Yaskawa INFORM job: A_ROOF_UPPER_0614_2_PAINT_44.JBI

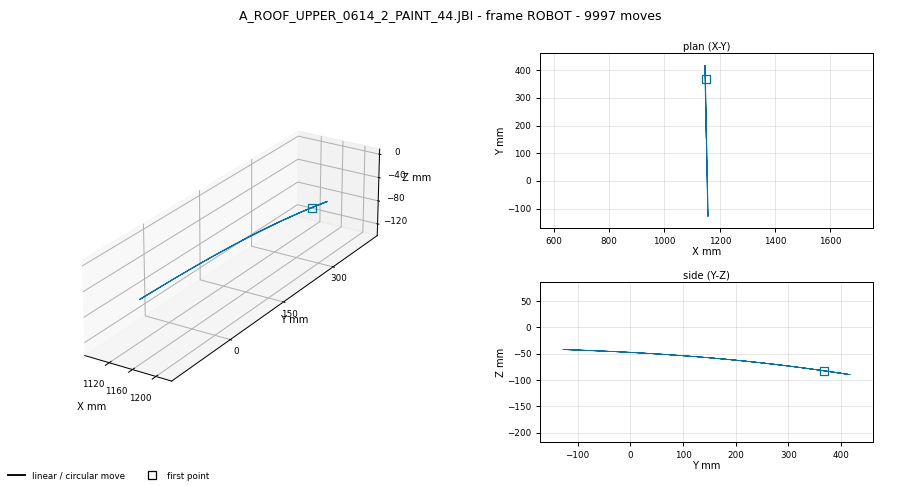
[picture p0: tool path of A_ROOF_UPPER_0614_2_PAINT_44.JBI in frame ROBOT, 9997 of 9997 moves have a stored position in this frame; points joined in program order, loops and branches not executed]
/JOB
//NAME A_ROOF_UPPER_0614_2_PAINT44
//POS
///NPOS 9997,0,0,0,0,0
///TOOL 1
///USER 0
///POSTYPE ROBOT
///RECTAN
///RCONF 1,0,0,0,0,0,0,0,0,0,0,0,0,0,0,0,0,0,0,0,0,0,0,0
C00000=1148.785,367.055,-82.178,-176.274,9.416,148.837
C00001=1148.782,367.302,-82.214,-176.271,9.420,148.837
C00002=1148.778,367.550,-82.249,-176.269,9.424,148.838
C00003=1148.773,367.797,-82.285,-176.266,9.428,148.838
C00004=1148.769,368.045,-82.321,-176.263,9.433,148.839
C00005=1148.766,368.292,-82.356,-176.261,9.436,148.839
C00006=1148.762,368.540,-82.392,-176.258,9.440,148.839
C00007=1148.758,368.787,-82.429,-176.256,9.445,148.840
C00008=1148.754,369.034,-82.464,-176.253,9.449,148.840
C00009=1148.751,369.282,-82.500,-176.250,9.453,148.841
C00010=1148.747,369.529,-82.535,-176.248,9.457,148.841
C00011=1148.742,369.776,-82.571,-176.246,9.461,148.841
C00012=1148.738,370.024,-82.607,-176.243,9.465,148.842
C00013=1148.735,370.271,-82.643,-176.241,9.470,148.842
C00014=1148.731,370.519,-82.679,-176.239,9.473,148.843
C00015=1148.727,370.766,-82.715,-176.236,9.477,148.843
C00016=1148.723,371.014,-82.750,-176.233,9.482,148.843
C00017=1148.719,371.261,-82.787,-176.231,9.486,148.844
C00018=1148.716,371.508,-82.823,-176.228,9.490,148.844
C00019=1148.712,371.756,-82.858,-176.226,9.494,148.845
C00020=1148.708,372.003,-82.895,-176.224,9.498,148.845
C00021=1148.704,372.250,-82.931,-176.221,9.503,148.846
C00022=1148.700,372.498,-82.966,-176.219,9.506,148.846
C00023=1148.696,372.745,-83.003,-176.217,9.510,148.846
C00024=1148.693,372.993,-83.039,-176.214,9.515,148.847
C00025=1148.689,373.240,-83.075,-176.212,9.519,148.847
C00026=1148.684,373.487,-83.111,-176.210,9.523,148.848
C00027=1148.680,373.734,-83.147,-176.208,9.527,148.848
C00028=1148.677,373.981,-83.183,-176.205,9.532,148.849
C00029=1148.673,374.229,-83.219,-176.203,9.535,148.849
C00030=1148.669,374.476,-83.255,-176.201,9.540,148.850
C00031=1148.665,374.724,-83.291,-176.199,9.543,148.850
C00032=1148.661,374.971,-83.328,-176.196,9.548,148.851
C00033=1148.657,375.218,-83.363,-176.194,9.553,148.851
C00034=1148.654,375.466,-83.401,-176.192,9.556,148.852
C00035=1148.651,375.713,-83.437,-176.190,9.561,148.852
C00036=1148.646,375.961,-83.473,-176.188,9.564,148.853
C00037=1148.643,376.208,-83.509,-176.186,9.569,148.853
C00038=1148.638,376.455,-83.545,-176.184,9.573,148.854
C00039=1148.635,376.702,-83.582,-176.182,9.577,148.854
C00040=1148.631,376.950,-83.618,-176.180,9.581,148.855
C00041=1148.627,377.197,-83.655,-176.179,9.585,148.855
C00042=1148.623,377.444,-83.691,-176.177,9.589,148.856
C00043=1148.619,377.692,-83.727,-176.175,9.593,148.856
C00044=1148.615,377.939,-83.763,-176.173,9.597,148.857
C00045=1148.611,378.186,-83.800,-176.171,9.601,148.858
C00046=1148.608,378.434,-83.836,-176.170,9.605,148.858
C00047=1148.604,378.681,-83.873,-176.168,9.609,148.859
C00048=1148.599,378.928,-83.909,-176.166,9.613,148.859
C00049=1148.596,379.175,-83.946,-176.164,9.617,148.860
C00050=1148.592,379.423,-83.982,-176.163,9.621,148.861
C00051=1148.588,379.670,-84.019,-176.161,9.625,148.861
C00052=1148.585,379.917,-84.055,-176.160,9.629,148.862
C00053=1148.581,380.165,-84.092,-176.158,9.633,148.863
C00054=1148.577,380.412,-84.129,-176.157,9.637,148.863
C00055=1148.573,380.659,-84.165,-176.156,9.641,148.864
C00056=1148.569,380.907,-84.201,-176.154,9.645,148.865
C00057=1148.565,381.154,-84.238,-176.153,9.648,148.865
C00058=1148.561,381.401,-84.275,-176.152,9.652,148.866
C00059=1148.557,381.648,-84.311,-176.151,9.656,148.867
C00060=1148.554,381.896,-84.349,-176.149,9.660,148.867
C00061=1148.550,382.143,-84.384,-176.149,9.663,148.868
C00062=1148.546,382.390,-84.421,-176.147,9.667,148.869
C00063=1148.542,382.638,-84.458,-176.147,9.671,148.869
C00064=1148.539,382.884,-84.494,-176.145,9.675,148.870
C00065=1148.535,383.132,-84.531,-176.145,9.678,148.871
C00066=1148.531,383.379,-84.568,-176.144,9.682,148.871
C00067=1148.527,383.627,-84.605,-176.143,9.685,148.872
C00068=1148.524,383.874,-84.641,-176.142,9.689,148.873
C00069=1148.520,384.121,-84.678,-176.142,9.692,148.874
C00070=1148.515,384.368,-84.715,-176.141,9.696,148.874
C00071=1148.511,384.615,-84.752,-176.140,9.700,148.875
C00072=1148.508,384.862,-84.788,-176.140,9.703,148.876
C00073=1148.505,385.110,-84.825,-176.139,9.706,148.877
C00074=1148.500,385.357,-84.862,-176.140,9.709,148.877
C00075=1148.496,385.604,-84.899,-176.139,9.712,148.878
C00076=1148.493,385.851,-84.935,-176.139,9.716,148.879
C00077=1148.489,386.098,-84.972,-176.138,9.719,148.880
C00078=1148.485,386.346,-85.009,-176.139,9.722,148.881
C00079=1148.481,386.593,-85.046,-176.138,9.725,148.881
C00080=1148.477,386.841,-85.083,-176.139,9.728,148.882
C00081=1148.474,387.088,-85.119,-176.138,9.732,148.883
C00082=1148.470,387.335,-85.156,-176.138,9.734,148.884
C00083=1148.466,387.583,-85.194,-176.138,9.738,148.885
C00084=1148.462,387.830,-85.230,-176.138,9.740,148.885
C00085=1148.458,388.077,-85.267,-176.139,9.743,148.886
C00086=1148.455,388.324,-85.304,-176.139,9.746,148.887
C00087=1148.451,388.571,-85.340,-176.139,9.749,148.888
C00088=1148.447,388.819,-85.378,-176.139,9.752,148.889
C00089=1148.443,389.066,-85.414,-176.140,9.755,148.889
C00090=1148.439,389.313,-85.451,-176.140,9.758,148.890
C00091=1148.436,389.560,-85.488,-176.141,9.761,148.891
C00092=1148.431,389.807,-85.524,-176.141,9.763,148.892
C00093=1148.428,390.055,-85.562,-176.141,9.766,148.893
C00094=1148.424,390.302,-85.599,-176.142,9.769,148.894
C00095=1148.420,390.549,-85.636,-176.143,9.771,148.895
C00096=1148.416,390.836,-85.678,-176.143,9.774,148.895
C00097=1148.411,391.123,-85.721,-176.144,9.777,148.896
C00098=1148.407,391.409,-85.764,-176.145,9.780,148.897
C00099=1148.402,391.696,-85.807,-176.145,9.783,148.898
C00100=1148.399,391.943,-85.843,-176.146,9.786,148.899
C00101=1148.395,392.190,-85.881,-176.146,9.789,148.900
C00102=1148.391,392.437,-85.918,-176.148,9.791,148.901
C00103=1148.387,392.684,-85.955,-176.148,9.793,148.902
C00104=1148.384,392.932,-85.992,-176.149,9.795,148.902
C00105=1148.380,393.179,-86.029,-176.149,9.798,148.903
C00106=1148.376,393.426,-86.065,-176.150,9.800,148.904
C00107=1148.372,393.674,-86.102,-176.151,9.802,148.905
C00108=1148.368,393.921,-86.139,-176.152,9.805,148.906
C00109=1148.365,394.168,-86.177,-176.153,9.807,148.907
C00110=1148.361,394.415,-86.214,-176.154,9.809,148.908
C00111=1148.357,394.662,-86.250,-176.155,9.812,148.909
C00112=1148.353,394.910,-86.287,-176.156,9.814,148.909
C00113=1148.350,395.157,-86.324,-176.157,9.816,148.910
C00114=1148.346,395.404,-86.361,-176.158,9.818,148.911
C00115=1148.342,395.652,-86.398,-176.159,9.821,148.912
C00116=1148.338,395.899,-86.435,-176.160,9.823,148.913
C00117=1148.334,396.146,-86.472,-176.160,9.825,148.913
C00118=1148.330,396.393,-86.509,-176.161,9.827,148.914
C00119=1148.326,396.640,-86.546,-176.163,9.829,148.915
C00120=1148.322,396.888,-86.583,-176.164,9.831,148.916
C00121=1148.319,397.134,-86.619,-176.165,9.833,148.917
C00122=1148.315,397.382,-86.657,-176.165,9.836,148.918
C00123=1148.311,397.630,-86.693,-176.166,9.838,148.918
C00124=1148.307,397.876,-86.731,-176.167,9.840,148.919
C00125=1148.303,398.123,-86.768,-176.169,9.842,148.920
C00126=1148.300,398.371,-86.805,-176.170,9.844,148.921
C00127=1148.296,398.618,-86.842,-176.171,9.846,148.922
C00128=1148.292,398.865,-86.878,-176.172,9.848,148.923
C00129=1148.288,399.112,-86.915,-176.173,9.851,148.924
C00130=1148.284,399.360,-86.952,-176.174,9.852,148.924
C00131=1148.281,399.607,-86.990,-176.175,9.854,148.925
C00132=1148.277,399.854,-87.027,-176.176,9.856,148.926
C00133=1148.273,400.101,-87.064,-176.177,9.858,148.927
C00134=1148.269,400.348,-87.100,-176.179,9.860,148.927
C00135=1148.265,400.596,-87.138,-176.180,9.862,148.928
C00136=1148.262,400.843,-87.174,-176.181,9.864,148.929
C00137=1148.258,401.090,-87.211,-176.182,9.866,148.930
C00138=1148.254,401.337,-87.248,-176.183,9.868,148.931
C00139=1148.251,401.585,-87.286,-176.184,9.870,148.931
C00140=1148.246,401.832,-87.322,-176.185,9.872,148.932
C00141=1148.242,402.079,-87.359,-176.186,9.874,148.933
C00142=1148.238,402.326,-87.396,-176.187,9.876,148.934
C00143=1148.234,402.574,-87.433,-176.188,9.878,148.935
C00144=1148.231,402.821,-87.470,-176.189,9.880,148.935
C00145=1148.228,403.068,-87.507,-176.191,9.881,148.936
C00146=1148.224,403.315,-87.544,-176.192,9.883,148.937
C00147=1148.219,403.562,-87.581,-176.192,9.885,148.938
C00148=1148.216,403.810,-87.618,-176.193,9.887,148.939
C00149=1148.212,404.057,-87.655,-176.195,9.889,148.939
C00150=1148.208,404.304,-87.692,-176.195,9.891,148.940
C00151=1148.204,404.551,-87.728,-176.196,9.893,148.941
C00152=1148.201,404.799,-87.766,-176.197,9.895,148.942
C00153=1148.197,405.046,-87.803,-176.198,9.897,148.942
C00154=1148.193,405.293,-87.840,-176.200,9.898,148.943
C00155=1148.189,405.540,-87.877,-176.201,9.900,148.944
C00156=1148.185,405.788,-87.914,-176.202,9.902,148.945
C00157=1148.181,406.035,-87.951,-176.203,9.904,148.945
C00158=1148.177,406.282,-87.988,-176.204,9.906,148.946
C00159=1148.174,406.529,-88.025,-176.204,9.907,148.947
C00160=1148.170,406.776,-88.061,-176.205,9.909,148.948
C00161=1148.167,407.024,-88.099,-176.206,9.911,148.948
C00162=1148.163,407.271,-88.135,-176.207,9.913,148.949
C00163=1148.158,407.518,-88.172,-176.208,9.915,148.950
C00164=1148.154,407.765,-88.209,-176.209,9.917,148.951
C00165=1148.151,408.013,-88.247,-176.210,9.919,148.951
C00166=1148.147,408.260,-88.284,-176.211,9.921,148.952
C00167=1148.144,408.507,-88.320,-176.212,9.922,148.953
C00168=1148.140,408.754,-88.357,-176.213,9.924,148.954
C00169=1148.136,409.002,-88.394,-176.214,9.926,148.954
C00170=1148.132,409.249,-88.431,-176.215,9.928,148.955
C00171=1148.128,409.496,-88.468,-176.216,9.930,148.956
C00172=1148.124,409.743,-88.506,-176.217,9.932,148.956
C00173=1148.121,409.991,-88.543,-176.218,9.934,148.957
C00174=1148.117,410.238,-88.580,-176.218,9.935,148.958
C00175=1148.113,410.485,-88.616,-176.219,9.937,148.959
C00176=1148.109,410.732,-88.653,-176.220,9.939,148.959
C00177=1148.105,410.979,-88.690,-176.221,9.941,148.960
C00178=1148.102,411.226,-88.728,-176.222,9.943,148.961
C00179=1148.098,411.474,-88.764,-176.222,9.946,148.962
C00180=1148.094,411.721,-88.801,-176.223,9.947,148.962
C00181=1148.090,411.968,-88.838,-176.224,9.949,148.963
C00182=1148.086,412.216,-88.875,-176.225,9.951,148.964
C00183=1148.082,412.463,-88.912,-176.225,9.953,148.964
C00184=1148.079,412.709,-88.949,-176.226,9.955,148.965
C00185=1148.075,412.956,-88.986,-176.227,9.957,148.966
C00186=1148.071,413.204,-89.023,-176.228,9.958,148.966
C00187=1148.067,413.452,-89.060,-176.229,9.961,148.967
C00188=1148.063,413.699,-89.097,-176.229,9.962,148.968
C00189=1148.059,413.946,-89.134,-176.229,9.965,148.969
C00190=1148.056,414.193,-89.172,-176.230,9.967,148.969
C00191=1148.052,414.440,-89.209,-176.231,9.969,148.970
C00192=1148.048,414.688,-89.246,-176.232,9.970,148.971
C00193=1148.045,414.935,-89.282,-176.233,9.972,148.971
C00194=1148.042,415.182,-89.320,-176.233,9.974,148.972
C00195=1148.040,415.429,-89.356,-176.234,9.977,148.973
C00196=1148.039,415.660,-89.390,-176.234,9.979,148.974
C00197=1148.039,415.890,-89.424,-176.235,9.980,148.974
C00198=1148.039,416.119,-89.458,-176.235,9.982,148.975
C00199=1148.040,416.350,-89.492,-176.236,9.983,148.975
C00200=1148.042,416.578,-89.526,-176.237,9.985,148.976
C00201=1148.044,416.809,-89.559,-176.237,9.987,148.977
C00202=1148.046,417.039,-89.593,-176.238,9.988,148.977
C00203=1148.050,417.267,-89.627,-176.238,9.990,148.978
C00204=1147.629,417.270,-89.676,-176.241,10.001,148.981
C00205=1147.626,417.038,-89.642,-176.240,9.999,148.980
C00206=1147.623,416.808,-89.609,-176.240,9.998,148.980
C00207=1147.621,416.576,-89.574,-176.239,9.996,148.979
C00208=1147.619,416.345,-89.540,-176.239,9.994,148.979
C00209=1147.619,416.113,-89.506,-176.238,9.992,148.978
C00210=1147.618,415.881,-89.472,-176.237,9.991,148.977
C00211=1147.619,415.649,-89.438,-176.237,9.989,148.977
C00212=1147.620,415.417,-89.403,-176.236,9.987,148.976
C00213=1147.622,415.171,-89.366,-176.235,9.985,148.976
C00214=1147.625,414.923,-89.329,-176.235,9.984,148.975
C00215=1147.627,414.676,-89.293,-176.235,9.981,148.974
C00216=1147.631,414.429,-89.255,-176.233,9.979,148.973
C00217=1147.635,414.182,-89.218,-176.233,9.977,148.973
C00218=1147.639,413.934,-89.181,-176.232,9.976,148.972
C00219=1147.643,413.687,-89.144,-176.231,9.973,148.971
C00220=1147.647,413.440,-89.107,-176.230,9.972,148.971
C00221=1147.651,413.193,-89.070,-176.230,9.969,148.970
C00222=1147.653,412.945,-89.033,-176.230,9.967,148.969
C00223=1147.658,412.698,-88.996,-176.228,9.965,148.968
C00224=1147.662,412.451,-88.960,-176.228,9.964,148.968
C00225=1147.666,412.204,-88.923,-176.227,9.962,148.967
C00226=1147.669,411.956,-88.885,-176.226,9.960,148.966
C00227=1147.673,411.709,-88.848,-176.225,9.958,148.966
C00228=1147.677,411.462,-88.811,-176.224,9.956,148.965
C00229=1147.681,411.215,-88.774,-176.224,9.954,148.964
C00230=1147.685,410.967,-88.737,-176.223,9.952,148.963
C00231=1147.688,410.720,-88.701,-176.222,9.950,148.963
C00232=1147.692,410.473,-88.664,-176.221,9.949,148.962
C00233=1147.696,410.226,-88.626,-176.220,9.947,148.961
C00234=1147.700,409.979,-88.589,-176.219,9.945,148.961
C00235=1147.704,409.731,-88.552,-176.218,9.943,148.960
C00236=1147.708,409.484,-88.515,-176.218,9.941,148.959
C00237=1147.712,409.237,-88.478,-176.217,9.939,148.958
C00238=1147.715,408.990,-88.441,-176.216,9.937,148.958
C00239=1147.719,408.743,-88.404,-176.215,9.935,148.957
C00240=1147.722,408.496,-88.367,-176.214,9.933,148.956
C00241=1147.726,408.248,-88.331,-176.213,9.931,148.955
C00242=1147.731,408.001,-88.294,-176.212,9.930,148.955
C00243=1147.734,407.753,-88.256,-176.211,9.927,148.954
C00244=1147.738,407.507,-88.219,-176.211,9.926,148.953
C00245=1147.742,407.260,-88.182,-176.209,9.924,148.952
C00246=1147.746,407.012,-88.145,-176.208,9.922,148.952
C00247=1147.749,406.765,-88.108,-176.208,9.920,148.951
C00248=1147.753,406.518,-88.072,-176.207,9.918,148.950
C00249=1147.757,406.270,-88.035,-176.206,9.916,148.950
C00250=1147.761,406.024,-87.997,-176.204,9.915,148.949
C00251=1147.764,405.776,-87.960,-176.203,9.913,148.948
C00252=1147.768,405.529,-87.923,-176.202,9.911,148.947
C00253=1147.772,405.282,-87.886,-176.201,9.909,148.946
C00254=1147.777,405.034,-87.849,-176.200,9.907,148.946
C00255=1147.780,404.787,-87.812,-176.200,9.905,148.945
C00256=1147.784,404.539,-87.775,-176.198,9.903,148.944
C00257=1147.787,404.293,-87.738,-176.197,9.901,148.943
C00258=1147.791,404.046,-87.702,-176.196,9.899,148.942
C00259=1147.795,403.799,-87.665,-176.195,9.898,148.942
C00260=1147.799,403.551,-87.627,-176.194,9.896,148.941
C00261=1147.803,403.304,-87.591,-176.193,9.894,148.940
C00262=1147.807,403.056,-87.554,-176.192,9.892,148.939
C00263=1147.811,402.810,-87.516,-176.191,9.890,148.939
C00264=1147.814,402.562,-87.479,-176.190,9.888,148.938
C00265=1147.818,402.315,-87.443,-176.189,9.886,148.937
C00266=1147.822,402.068,-87.406,-176.188,9.884,148.936
C00267=1147.826,401.821,-87.369,-176.187,9.882,148.935
C00268=1147.829,401.573,-87.332,-176.185,9.881,148.935
C00269=1147.833,401.326,-87.294,-176.184,9.879,148.934
C00270=1147.837,401.079,-87.257,-176.183,9.877,148.933
C00271=1147.841,400.832,-87.220,-176.182,9.875,148.932
C00272=1147.845,400.584,-87.183,-176.181,9.873,148.931
C00273=1147.848,400.337,-87.147,-176.180,9.871,148.931
C00274=1147.852,400.090,-87.110,-176.179,9.868,148.930
C00275=1147.856,399.843,-87.072,-176.178,9.867,148.929
C00276=1147.860,399.595,-87.035,-176.177,9.865,148.928
C00277=1147.864,399.348,-86.998,-176.176,9.863,148.927
C00278=1147.868,399.101,-86.962,-176.175,9.861,148.927
C00279=1147.872,398.854,-86.925,-176.174,9.859,148.926
C00280=1147.876,398.607,-86.888,-176.173,9.856,148.925
C00281=1147.879,398.359,-86.851,-176.171,9.854,148.924
C00282=1147.882,398.113,-86.814,-176.170,9.852,148.923
C00283=1147.887,397.865,-86.777,-176.169,9.850,148.922
C00284=1147.891,397.618,-86.740,-176.168,9.848,148.922
C00285=1147.894,397.370,-86.703,-176.167,9.846,148.921
C00286=1147.898,397.123,-86.666,-176.166,9.844,148.920
C00287=1147.902,396.876,-86.629,-176.165,9.842,148.919
C00288=1147.906,396.629,-86.591,-176.164,9.840,148.918
C00289=1147.909,396.382,-86.555,-176.163,9.838,148.918
C00290=1147.913,396.135,-86.518,-176.162,9.836,148.917
C00291=1147.917,395.887,-86.481,-176.161,9.834,148.916
C00292=1147.921,395.640,-86.444,-176.160,9.831,148.915
C00293=1147.925,395.392,-86.407,-176.159,9.829,148.914
C00294=1147.929,395.145,-86.370,-176.158,9.827,148.913
C00295=1147.933,394.899,-86.333,-176.157,9.825,148.913
C00296=1147.937,394.651,-86.296,-176.157,9.822,148.912
C00297=1147.940,394.404,-86.259,-176.155,9.820,148.911
C00298=1147.943,394.157,-86.222,-176.154,9.818,148.910
C00299=1147.948,393.909,-86.185,-176.153,9.816,148.909
C00300=1147.952,393.662,-86.148,-176.153,9.813,148.908
C00301=1147.956,393.415,-86.112,-176.152,9.811,148.907
C00302=1147.959,393.168,-86.074,-176.151,9.808,148.907
C00303=1147.963,392.921,-86.037,-176.150,9.806,148.906
C00304=1147.966,392.674,-86.001,-176.150,9.804,148.905
C00305=1147.970,392.426,-85.964,-176.149,9.801,148.904
C00306=1147.974,392.179,-85.926,-176.148,9.799,148.903
C00307=1147.978,391.931,-85.890,-176.147,9.797,148.902
C00308=1147.982,391.684,-85.853,-176.147,9.794,148.901
C00309=1147.986,391.398,-85.810,-176.146,9.791,148.901
C00310=1147.991,391.111,-85.767,-176.145,9.788,148.900
C00311=1147.996,390.825,-85.724,-176.145,9.785,148.899
C00312=1148.000,390.538,-85.681,-176.144,9.782,148.898
C00313=1148.003,390.290,-85.644,-176.143,9.780,148.897
C00314=1148.007,390.043,-85.608,-176.142,9.777,148.896
C00315=1148.011,389.796,-85.571,-176.142,9.774,148.895
C00316=1148.015,389.549,-85.534,-176.142,9.772,148.894
C00317=1148.018,389.302,-85.496,-176.141,9.769,148.894
C00318=1148.022,389.054,-85.459,-176.141,9.766,148.893
C00319=1148.026,388.807,-85.422,-176.141,9.763,148.892
C00320=1148.030,388.560,-85.386,-176.140,9.760,148.891
C00321=1148.034,388.313,-85.349,-176.140,9.758,148.890
C00322=1148.037,388.065,-85.312,-176.140,9.754,148.889
C00323=1148.041,387.818,-85.275,-176.140,9.752,148.889
C00324=1148.045,387.571,-85.238,-176.139,9.749,148.888
C00325=1148.049,387.324,-85.202,-176.140,9.745,148.887
C00326=1148.053,387.077,-85.165,-176.139,9.742,148.886
C00327=1148.056,386.829,-85.128,-176.139,9.740,148.885
C00328=1148.061,386.582,-85.091,-176.139,9.736,148.884
C00329=1148.065,386.335,-85.054,-176.140,9.733,148.884
C00330=1148.068,386.088,-85.018,-176.140,9.730,148.883
C00331=1148.071,385.840,-84.981,-176.140,9.727,148.882
C00332=1148.076,385.593,-84.944,-176.140,9.723,148.881
C00333=1148.080,385.345,-84.907,-176.140,9.721,148.881
C00334=1148.084,385.098,-84.870,-176.141,9.717,148.880
C00335=1148.087,384.851,-84.834,-176.141,9.714,148.879
C00336=1148.091,384.604,-84.797,-176.142,9.710,148.878
C00337=1148.095,384.356,-84.760,-176.142,9.707,148.878
C00338=1148.099,384.109,-84.723,-176.143,9.704,148.877
C00339=1148.102,383.862,-84.687,-176.144,9.700,148.876
C00340=1148.106,383.615,-84.650,-176.145,9.696,148.875
C00341=1148.110,383.368,-84.613,-176.145,9.693,148.875
C00342=1148.114,383.121,-84.576,-176.146,9.689,148.874
C00343=1148.117,382.873,-84.540,-176.147,9.686,148.873
C00344=1148.121,382.626,-84.503,-176.147,9.682,148.873
C00345=1148.125,382.379,-84.466,-176.149,9.678,148.872
C00346=1148.129,382.131,-84.429,-176.150,9.674,148.871
C00347=1148.133,381.885,-84.393,-176.151,9.671,148.871
C00348=1148.137,381.637,-84.356,-176.152,9.667,148.870
C00349=1148.141,381.389,-84.319,-176.153,9.663,148.869
C00350=1148.144,381.142,-84.283,-176.155,9.659,148.869
C00351=1148.148,380.895,-84.246,-176.155,9.656,148.868
C00352=1148.152,380.648,-84.209,-176.157,9.652,148.867
C00353=1148.156,380.401,-84.173,-176.158,9.648,148.867
C00354=1148.160,380.154,-84.136,-176.160,9.644,148.866
C00355=1148.164,379.906,-84.100,-176.161,9.640,148.865
C00356=1148.167,379.659,-84.064,-176.163,9.636,148.865
C00357=1148.172,379.412,-84.027,-176.164,9.633,148.864
C00358=1148.175,379.164,-83.990,-176.166,9.629,148.863
C00359=1148.178,378.917,-83.954,-176.168,9.624,148.863
C00360=1148.183,378.669,-83.917,-176.169,9.620,148.862
C00361=1148.186,378.422,-83.881,-176.171,9.616,148.862
C00362=1148.190,378.175,-83.844,-176.173,9.613,148.861
C00363=1148.195,377.927,-83.808,-176.175,9.608,148.860
C00364=1148.198,377.680,-83.772,-176.176,9.604,148.860
C00365=1148.202,377.433,-83.735,-176.178,9.600,148.859
C00366=1148.206,377.186,-83.699,-176.180,9.596,148.859
C00367=1148.210,376.938,-83.663,-176.182,9.592,148.858
C00368=1148.214,376.691,-83.626,-176.184,9.588,148.858
C00369=1148.218,376.444,-83.590,-176.186,9.584,148.857
C00370=1148.222,376.197,-83.553,-176.188,9.580,148.857
C00371=1148.225,375.950,-83.517,-176.190,9.576,148.856
C00372=1148.229,375.702,-83.481,-176.192,9.572,148.856
C00373=1148.233,375.455,-83.445,-176.194,9.567,148.855
C00374=1148.237,375.207,-83.409,-176.197,9.563,148.855
C00375=1148.241,374.960,-83.372,-176.199,9.559,148.854
C00376=1148.245,374.712,-83.336,-176.201,9.555,148.854
C00377=1148.248,374.465,-83.299,-176.203,9.551,148.853
C00378=1148.252,374.217,-83.263,-176.205,9.547,148.853
C00379=1148.256,373.970,-83.227,-176.208,9.542,148.852
C00380=1148.260,373.722,-83.191,-176.209,9.539,148.852
C00381=1148.263,373.476,-83.155,-176.212,9.534,148.851
C00382=1148.268,373.229,-83.119,-176.214,9.530,148.851
C00383=1148.272,372.982,-83.083,-176.216,9.526,148.850
C00384=1148.275,372.734,-83.047,-176.219,9.522,148.850
C00385=1148.280,372.486,-83.011,-176.221,9.518,148.849
C00386=1148.283,372.239,-82.975,-176.224,9.513,148.849
C00387=1148.287,371.992,-82.939,-176.226,9.510,148.849
C00388=1148.291,371.745,-82.902,-176.228,9.505,148.848
C00389=1148.294,371.497,-82.867,-176.231,9.501,148.848
C00390=1148.299,371.249,-82.831,-176.233,9.496,148.847
C00391=1148.303,371.002,-82.795,-176.235,9.493,148.847
C00392=1148.306,370.755,-82.759,-176.238,9.489,148.846
C00393=1148.310,370.507,-82.723,-176.240,9.484,148.846
C00394=1148.314,370.260,-82.687,-176.243,9.480,148.845
C00395=1148.317,370.013,-82.651,-176.246,9.476,148.845
C00396=1148.322,369.765,-82.615,-176.248,9.472,148.845
C00397=1148.325,369.517,-82.579,-176.250,9.468,148.844
C00398=1148.330,369.271,-82.544,-176.253,9.464,148.844
C00399=1148.333,369.023,-82.508,-176.256,9.459,148.844
C00400=1148.337,368.776,-82.472,-176.258,9.455,148.843
C00401=1148.341,368.528,-82.436,-176.260,9.452,148.843
C00402=1148.345,368.281,-82.400,-176.263,9.447,148.842
C00403=1148.349,368.033,-82.364,-176.265,9.443,148.842
C00404=1148.353,367.786,-82.329,-176.268,9.439,148.842
C00405=1148.356,367.538,-82.293,-176.271,9.434,148.841
C00406=1148.361,367.291,-82.258,-176.273,9.431,148.841
C00407=1148.364,367.044,-82.222,-176.276,9.427,148.841
C00408=1148.369,366.796,-82.186,-176.279,9.423,148.840
C00409=1148.372,366.549,-82.151,-176.281,9.418,148.840
C00410=1148.376,366.301,-82.115,-176.284,9.414,148.840
C00411=1148.380,366.054,-82.080,-176.287,9.410,148.839
C00412=1148.384,365.807,-82.045,-176.289,9.407,148.839
C00413=1148.388,365.523,-82.004,-176.292,9.401,148.838
C00414=1148.393,365.240,-81.963,-176.295,9.397,148.838
C00415=1148.397,364.957,-81.922,-176.298,9.392,148.838
C00416=1148.402,364.673,-81.881,-176.301,9.388,148.837
C00417=1148.405,364.426,-81.846,-176.303,9.384,148.837
C00418=1148.410,364.179,-81.811,-176.306,9.379,148.837
C00419=1148.413,363.931,-81.775,-176.309,9.375,148.836
C00420=1148.417,363.684,-81.740,-176.311,9.372,148.836
C00421=1148.421,363.436,-81.705,-176.314,9.367,148.835
C00422=1148.425,363.189,-81.670,-176.316,9.363,148.835
C00423=1148.429,362.942,-81.634,-176.319,9.359,148.835
C00424=1148.433,362.694,-81.598,-176.321,9.356,148.834
C00425=1148.437,362.446,-81.562,-176.324,9.352,148.834
C00426=1148.441,362.199,-81.528,-176.327,9.347,148.834
C00427=1148.445,361.951,-81.492,-176.330,9.343,148.833
C00428=1148.449,361.704,-81.457,-176.331,9.340,148.833
C00429=1148.452,361.457,-81.422,-176.334,9.335,148.833
C00430=1148.456,361.209,-81.387,-176.337,9.331,148.832
C00431=1148.460,360.962,-81.352,-176.340,9.327,148.832
C00432=1148.464,360.714,-81.316,-176.342,9.324,148.832
C00433=1148.468,360.467,-81.282,-176.345,9.319,148.831
C00434=1148.472,360.219,-81.246,-176.347,9.315,148.831
C00435=1148.476,359.971,-81.211,-176.349,9.312,148.831
C00436=1148.479,359.724,-81.176,-176.352,9.308,148.830
C00437=1148.484,359.477,-81.141,-176.355,9.303,148.830
C00438=1148.488,359.229,-81.106,-176.357,9.300,148.830
C00439=1148.491,358.981,-81.070,-176.360,9.296,148.830
C00440=1148.496,358.734,-81.036,-176.363,9.291,148.829
C00441=1148.500,358.486,-81.000,-176.365,9.288,148.829
C00442=1148.503,358.239,-80.966,-176.367,9.284,148.828
C00443=1148.507,357.992,-80.931,-176.370,9.280,148.828
C00444=1148.511,357.744,-80.896,-176.373,9.276,148.828
C00445=1148.515,357.497,-80.861,-176.375,9.272,148.827
C00446=1148.519,357.249,-80.826,-176.378,9.268,148.827
C00447=1148.523,357.001,-80.790,-176.380,9.264,148.827
C00448=1148.528,356.754,-80.756,-176.383,9.260,148.826
C00449=1148.530,356.507,-80.721,-176.385,9.257,148.826
C00450=1148.535,356.259,-80.687,-176.388,9.253,148.826
C00451=1148.539,356.011,-80.652,-176.391,9.248,148.826
C00452=1148.543,355.763,-80.616,-176.392,9.245,148.825
C00453=1148.546,355.516,-80.582,-176.395,9.241,148.825
C00454=1148.550,355.268,-80.547,-176.398,9.238,148.825
C00455=1148.555,355.021,-80.512,-176.400,9.233,148.824
C00456=1148.559,354.773,-80.477,-176.403,9.229,148.824
C00457=1148.563,354.526,-80.444,-176.405,9.225,148.824
C00458=1148.566,354.279,-80.408,-176.408,9.221,148.823
C00459=1148.570,354.031,-80.373,-176.410,9.218,148.823
C00460=1148.575,353.783,-80.339,-176.413,9.214,148.823
C00461=1148.578,353.535,-80.305,-176.416,9.210,148.822
C00462=1148.582,353.289,-80.269,-176.417,9.206,148.822
C00463=1148.586,353.040,-80.234,-176.420,9.202,148.822
C00464=1148.590,352.793,-80.201,-176.423,9.199,148.821
C00465=1148.594,352.545,-80.166,-176.425,9.194,148.821
C00466=1148.599,352.298,-80.131,-176.428,9.190,148.821
C00467=1148.602,352.050,-80.097,-176.430,9.187,148.821
C00468=1148.606,351.803,-80.062,-176.433,9.183,148.820
C00469=1148.610,351.555,-80.027,-176.435,9.179,148.820
C00470=1148.614,351.308,-79.993,-176.438,9.175,148.820
C00471=1148.618,351.060,-79.958,-176.440,9.172,148.819
C00472=1148.622,350.812,-79.924,-176.443,9.168,148.819
C00473=1148.626,350.565,-79.890,-176.446,9.163,148.819
C00474=1148.630,350.317,-79.855,-176.448,9.160,148.818
C00475=1148.634,350.070,-79.821,-176.451,9.156,148.818
C00476=1148.638,349.822,-79.786,-176.453,9.152,148.818
C00477=1148.642,349.575,-79.753,-176.455,9.148,148.817
C00478=1148.646,349.327,-79.718,-176.458,9.145,148.817
C00479=1148.650,349.079,-79.683,-176.461,9.141,148.817
C00480=1148.654,348.832,-79.649,-176.463,9.136,148.816
C00481=1148.658,348.584,-79.615,-176.466,9.133,148.816
C00482=1148.662,348.337,-79.581,-176.468,9.129,148.816
C00483=1148.666,348.089,-79.546,-176.470,9.125,148.816
C00484=1148.670,347.842,-79.512,-176.473,9.121,148.815
C00485=1148.674,347.593,-79.478,-176.476,9.118,148.815
C00486=1148.678,347.346,-79.444,-176.478,9.114,148.815
C00487=1148.682,347.098,-79.410,-176.480,9.110,148.815
C00488=1148.686,346.851,-79.375,-176.483,9.106,148.814
C00489=1148.690,346.603,-79.341,-176.486,9.102,148.814
C00490=1148.694,346.355,-79.307,-176.488,9.099,148.814
C00491=1148.698,346.108,-79.273,-176.491,9.095,148.813
C00492=1148.702,345.860,-79.239,-176.493,9.091,148.813
C00493=1148.705,345.612,-79.205,-176.496,9.087,148.813
C00494=1148.710,345.365,-79.170,-176.498,9.084,148.812
C00495=1148.714,345.117,-79.137,-176.501,9.079,148.812
C00496=1148.718,344.869,-79.102,-176.503,9.076,148.812
C00497=1148.722,344.622,-79.068,-176.506,9.072,148.812
C00498=1148.726,344.374,-79.035,-176.508,9.069,148.811
C00499=1148.730,344.126,-79.000,-176.511,9.064,148.811
C00500=1148.734,343.879,-78.967,-176.513,9.061,148.811
C00501=1148.738,343.631,-78.933,-176.516,9.057,148.810
C00502=1148.743,343.384,-78.899,-176.518,9.054,148.810
C00503=1148.746,343.136,-78.865,-176.521,9.049,148.810
C00504=1148.750,342.888,-78.832,-176.523,9.046,148.810
C00505=1148.755,342.641,-78.797,-176.526,9.042,148.810
C00506=1148.758,342.393,-78.764,-176.529,9.038,148.809
C00507=1148.762,342.146,-78.730,-176.531,9.034,148.809
C00508=1148.767,341.897,-78.696,-176.534,9.030,148.809
C00509=1148.771,341.650,-78.662,-176.536,9.027,148.808
C00510=1148.774,341.402,-78.629,-176.539,9.023,148.808
C00511=1148.778,341.155,-78.595,-176.541,9.019,148.808
C00512=1148.783,340.907,-78.561,-176.544,9.015,148.808
C00513=1148.787,340.660,-78.527,-176.546,9.012,148.807
C00514=1148.790,340.411,-78.494,-176.549,9.008,148.807
C00515=1148.794,340.164,-78.460,-176.551,9.004,148.807
C00516=1148.799,339.916,-78.426,-176.554,9.000,148.806
C00517=1148.803,339.636,-78.388,-176.557,8.996,148.806
C00518=1148.808,339.356,-78.350,-176.560,8.992,148.806
C00519=1148.812,339.076,-78.312,-176.563,8.988,148.806
C00520=1148.817,338.795,-78.274,-176.565,8.984,148.805
C00521=1148.821,338.547,-78.240,-176.568,8.980,148.805
C00522=1148.825,338.300,-78.207,-176.571,8.976,148.805
C00523=1148.829,338.052,-78.173,-176.573,8.973,148.805
C00524=1148.833,337.805,-78.140,-176.576,8.969,148.804
C00525=1148.836,337.557,-78.106,-176.578,8.966,148.804
C00526=1148.841,337.309,-78.073,-176.581,8.961,148.804
C00527=1148.846,337.061,-78.039,-176.583,8.958,148.804
C00528=1148.850,336.813,-78.006,-176.586,8.954,148.803
C00529=1148.853,336.566,-77.972,-176.588,8.951,148.803
C00530=1148.858,336.319,-77.939,-176.591,8.946,148.803
C00531=1148.861,336.070,-77.905,-176.593,8.943,148.803
C00532=1148.865,335.822,-77.872,-176.596,8.939,148.802
C00533=1148.869,335.575,-77.839,-176.599,8.936,148.802
C00534=1148.874,335.327,-77.806,-176.601,8.931,148.802
C00535=1148.877,335.080,-77.772,-176.603,8.928,148.802
C00536=1148.882,334.832,-77.739,-176.606,8.925,148.801
C00537=1148.886,334.584,-77.706,-176.609,8.921,148.801
C00538=1148.890,334.337,-77.673,-176.611,8.918,148.801
C00539=1148.893,334.088,-77.639,-176.614,8.913,148.801
C00540=1148.897,333.840,-77.606,-176.616,8.910,148.800
C00541=1148.902,333.593,-77.573,-176.619,8.906,148.800
C00542=1148.906,333.345,-77.540,-176.621,8.903,148.800
C00543=1148.910,333.097,-77.506,-176.624,8.898,148.800
C00544=1148.914,332.850,-77.473,-176.626,8.895,148.799
C00545=1148.918,332.602,-77.440,-176.629,8.891,148.799
C00546=1148.922,332.354,-77.407,-176.631,8.888,148.799
C00547=1148.926,332.106,-77.374,-176.634,8.885,148.799
C00548=1148.931,331.859,-77.341,-176.637,8.880,148.798
C00549=1148.935,331.611,-77.307,-176.639,8.877,148.798
C00550=1148.938,331.363,-77.275,-176.642,8.873,148.798
C00551=1148.942,331.116,-77.242,-176.644,8.870,148.798
C00552=1148.946,330.868,-77.209,-176.647,8.866,148.798
C00553=1148.951,330.620,-77.175,-176.650,8.862,148.797
C00554=1148.955,330.372,-77.143,-176.652,8.859,148.797
C00555=1148.959,330.124,-77.110,-176.655,8.855,148.797
C00556=1148.963,329.876,-77.077,-176.657,8.852,148.797
C00557=1148.967,329.629,-77.044,-176.660,8.848,148.797
C00558=1148.971,329.381,-77.011,-176.662,8.844,148.796
C00559=1148.975,329.134,-76.978,-176.665,8.840,148.796
C00560=1148.979,328.885,-76.945,-176.668,8.837,148.796
C00561=1148.984,328.638,-76.912,-176.670,8.834,148.796
C00562=1148.988,328.390,-76.879,-176.673,8.830,148.795
C00563=1148.991,328.142,-76.846,-176.675,8.826,148.795
C00564=1148.996,327.894,-76.814,-176.678,8.822,148.795
C00565=1149.000,327.646,-76.781,-176.680,8.819,148.795
C00566=1149.004,327.399,-76.748,-176.683,8.815,148.794
C00567=1149.007,327.151,-76.716,-176.685,8.811,148.794
C00568=1149.012,326.903,-76.683,-176.687,8.808,148.794
C00569=1149.016,326.655,-76.650,-176.690,8.804,148.794
C00570=1149.020,326.407,-76.617,-176.693,8.801,148.794
C00571=1149.024,326.159,-76.585,-176.696,8.797,148.794
C00572=1149.028,325.912,-76.551,-176.698,8.794,148.793
C00573=1149.032,325.663,-76.519,-176.701,8.791,148.793
C00574=1149.036,325.416,-76.486,-176.704,8.786,148.793
C00575=1149.041,325.168,-76.454,-176.706,8.783,148.793
C00576=1149.045,324.920,-76.421,-176.709,8.779,148.793
C00577=1149.048,324.672,-76.389,-176.711,8.776,148.792
C00578=1149.053,324.425,-76.356,-176.713,8.773,148.792
C00579=1149.057,324.176,-76.324,-176.716,8.768,148.792
C00580=1149.060,323.929,-76.291,-176.719,8.765,148.792
C00581=1149.065,323.681,-76.259,-176.721,8.762,148.792
C00582=1149.068,323.433,-76.226,-176.724,8.758,148.791
C00583=1149.073,323.185,-76.194,-176.726,8.755,148.791
C00584=1149.077,322.938,-76.161,-176.729,8.750,148.791
C00585=1149.081,322.690,-76.129,-176.731,8.747,148.791
C00586=1149.085,322.442,-76.096,-176.734,8.744,148.790
C00587=1149.089,322.194,-76.064,-176.737,8.740,148.790
C00588=1149.093,321.946,-76.032,-176.739,8.737,148.790
C00589=1149.097,321.698,-75.999,-176.742,8.732,148.790
C00590=1149.101,321.450,-75.967,-176.745,8.730,148.790
C00591=1149.106,321.202,-75.935,-176.747,8.726,148.790
C00592=1149.110,320.955,-75.902,-176.750,8.722,148.789
C00593=1149.113,320.707,-75.870,-176.752,8.719,148.789
C00594=1149.118,320.458,-75.838,-176.755,8.716,148.789
C00595=1149.121,320.211,-75.805,-176.757,8.712,148.789
C00596=1149.126,319.963,-75.773,-176.760,8.708,148.789
C00597=1149.130,319.715,-75.741,-176.762,8.705,148.788
C00598=1149.135,319.467,-75.709,-176.765,8.701,148.788
C00599=1149.138,319.219,-75.677,-176.767,8.698,148.788
C00600=1149.142,318.971,-75.644,-176.770,8.695,148.788
C00601=1149.147,318.724,-75.612,-176.773,8.691,148.788
C00602=1149.150,318.476,-75.581,-176.775,8.687,148.788
C00603=1149.155,318.227,-75.548,-176.778,8.683,148.787
C00604=1149.159,317.979,-75.516,-176.781,8.680,148.787
C00605=1149.163,317.732,-75.483,-176.783,8.677,148.787
C00606=1149.167,317.484,-75.452,-176.786,8.673,148.787
C00607=1149.171,317.236,-75.420,-176.789,8.670,148.787
C00608=1149.175,316.988,-75.387,-176.791,8.666,148.787
C00609=1149.179,316.741,-75.356,-176.794,8.662,148.786
C00610=1149.184,316.492,-75.323,-176.796,8.659,148.786
C00611=1149.188,316.244,-75.292,-176.798,8.656,148.786
C00612=1149.192,315.997,-75.260,-176.801,8.652,148.786
C00613=1149.196,315.749,-75.228,-176.804,8.649,148.786
C00614=1149.200,315.500,-75.196,-176.806,8.645,148.786
C00615=1149.204,315.253,-75.164,-176.809,8.641,148.785
C00616=1149.208,315.005,-75.132,-176.812,8.638,148.785
C00617=1149.212,314.757,-75.100,-176.814,8.635,148.785
C00618=1149.217,314.509,-75.069,-176.817,8.631,148.785
C00619=1149.221,314.261,-75.037,-176.820,8.628,148.785
C00620=1149.225,314.013,-75.004,-176.822,8.625,148.785
C00621=1149.229,313.735,-74.969,-176.825,8.620,148.784
C00622=1149.234,313.458,-74.934,-176.828,8.616,148.784
C00623=1149.239,313.181,-74.899,-176.831,8.612,148.784
C00624=1149.244,312.903,-74.862,-176.834,8.608,148.784
C00625=1149.248,312.655,-74.830,-176.836,8.605,148.784
C00626=1149.252,312.407,-74.799,-176.839,8.602,148.784
C00627=1149.256,312.159,-74.767,-176.842,8.598,148.783
C00628=1149.260,311.911,-74.736,-176.844,8.595,148.783
C00629=1149.265,311.663,-74.704,-176.847,8.592,148.783
C00630=1149.268,311.415,-74.672,-176.849,8.588,148.783
C00631=1149.273,311.168,-74.641,-176.852,8.584,148.783
C00632=1149.277,310.919,-74.609,-176.855,8.581,148.783
C00633=1149.280,310.671,-74.578,-176.857,8.578,148.783
C00634=1149.285,310.424,-74.546,-176.860,8.574,148.782
C00635=1149.288,310.176,-74.514,-176.862,8.571,148.782
C00636=1149.294,309.927,-74.483,-176.865,8.568,148.782
C00637=1149.297,309.679,-74.451,-176.868,8.564,148.782
C00638=1149.302,309.432,-74.420,-176.870,8.560,148.782
C00639=1149.306,309.183,-74.388,-176.873,8.557,148.782
C00640=1149.309,308.935,-74.357,-176.875,8.554,148.782
C00641=1149.314,308.687,-74.326,-176.878,8.550,148.781
C00642=1149.318,308.439,-74.294,-176.881,8.547,148.781
C00643=1149.322,308.192,-74.263,-176.883,8.544,148.781
C00644=1149.326,307.943,-74.231,-176.886,8.540,148.781
C00645=1149.330,307.696,-74.200,-176.889,8.537,148.781
C00646=1149.334,307.447,-74.169,-176.891,8.533,148.781
C00647=1149.339,307.200,-74.137,-176.894,8.530,148.781
C00648=1149.343,306.951,-74.106,-176.897,8.526,148.780
C00649=1149.347,306.704,-74.075,-176.899,8.523,148.780
C00650=1149.351,306.455,-74.044,-176.902,8.520,148.780
C00651=1149.355,306.208,-74.012,-176.905,8.516,148.780
C00652=1149.359,305.959,-73.981,-176.907,8.513,148.780
C00653=1149.364,305.712,-73.950,-176.909,8.509,148.780
C00654=1149.368,305.463,-73.918,-176.912,8.506,148.780
C00655=1149.372,305.216,-73.887,-176.915,8.502,148.780
C00656=1149.377,304.968,-73.856,-176.917,8.499,148.779
C00657=1149.381,304.719,-73.825,-176.920,8.496,148.779
C00658=1149.385,304.472,-73.794,-176.922,8.493,148.779
C00659=1149.389,304.223,-73.762,-176.925,8.489,148.779
C00660=1149.394,303.975,-73.732,-176.928,8.486,148.779
C00661=1149.397,303.727,-73.700,-176.930,8.483,148.779
C00662=1149.402,303.479,-73.669,-176.933,8.479,148.779
C00663=1149.407,303.231,-73.638,-176.936,8.476,148.779
C00664=1149.410,302.983,-73.606,-176.938,8.472,148.778
C00665=1149.415,302.735,-73.576,-176.941,8.469,148.779
C00666=1149.418,302.487,-73.545,-176.943,8.466,148.778
C00667=1149.423,302.239,-73.514,-176.946,8.462,148.778
C00668=1149.427,301.992,-73.483,-176.949,8.459,148.778
C00669=1149.431,301.743,-73.452,-176.951,8.456,148.778
C00670=1149.436,301.495,-73.421,-176.954,8.452,148.778
C00671=1149.440,301.246,-73.390,-176.957,8.449,148.778
C00672=1149.444,300.999,-73.360,-176.959,8.445,148.778
C00673=1149.448,300.751,-73.328,-176.962,8.442,148.778
C00674=1149.452,300.503,-73.297,-176.964,8.439,148.777
C00675=1149.456,300.255,-73.266,-176.967,8.435,148.777
C00676=1149.461,300.007,-73.236,-176.970,8.432,148.777
C00677=1149.464,299.758,-73.205,-176.972,8.429,148.777
C00678=1149.469,299.511,-73.174,-176.975,8.426,148.777
C00679=1149.474,299.263,-73.143,-176.978,8.422,148.777
C00680=1149.478,299.014,-73.112,-176.980,8.419,148.777
C00681=1149.481,298.766,-73.082,-176.983,8.416,148.777
C00682=1149.486,298.518,-73.051,-176.986,8.412,148.777
C00683=1149.490,298.270,-73.020,-176.988,8.409,148.777
C00684=1149.494,298.022,-72.990,-176.991,8.405,148.776
C00685=1149.499,297.774,-72.959,-176.994,8.402,148.776
C00686=1149.503,297.525,-72.928,-176.996,8.399,148.776
C00687=1149.506,297.278,-72.898,-176.999,8.396,148.776
C00688=1149.511,297.030,-72.867,-177.001,8.393,148.776
C00689=1149.516,296.782,-72.837,-177.004,8.389,148.776
C00690=1149.519,296.533,-72.806,-177.007,8.386,148.776
C00691=1149.524,296.286,-72.775,-177.009,8.383,148.776
C00692=1149.528,296.038,-72.744,-177.012,8.380,148.776
C00693=1149.532,295.790,-72.714,-177.015,8.376,148.776
C00694=1149.536,295.541,-72.683,-177.018,8.373,148.776
C00695=1149.540,295.293,-72.654,-177.020,8.369,148.775
C00696=1149.545,295.045,-72.623,-177.023,8.366,148.776
C00697=1149.550,294.797,-72.592,-177.025,8.363,148.775
C00698=1149.553,294.549,-72.562,-177.028,8.359,148.775
C00699=1149.557,294.301,-72.531,-177.031,8.356,148.775
C00700=1149.561,294.053,-72.501,-177.033,8.353,148.775
C00701=1149.566,293.805,-72.471,-177.036,8.350,148.775
C00702=1149.569,293.556,-72.440,-177.038,8.347,148.775
C00703=1149.574,293.308,-72.409,-177.042,8.343,148.775
C00704=1149.578,293.061,-72.379,-177.044,8.340,148.775
C00705=1149.583,292.812,-72.349,-177.047,8.337,148.775
C00706=1149.587,292.564,-72.319,-177.049,8.333,148.775
C00707=1149.591,292.316,-72.288,-177.052,8.330,148.775
C00708=1149.595,292.067,-72.258,-177.054,8.327,148.774
C00709=1149.600,291.819,-72.228,-177.058,8.323,148.774
C00710=1149.603,291.572,-72.197,-177.060,8.320,148.774
C00711=1149.608,291.323,-72.167,-177.063,8.317,148.774
C00712=1149.612,291.076,-72.137,-177.065,8.314,148.774
C00713=1149.616,290.827,-72.107,-177.068,8.311,148.774
C00714=1149.620,290.579,-72.077,-177.071,8.307,148.774
C00715=1149.624,290.331,-72.047,-177.073,8.304,148.774
C00716=1149.629,290.082,-72.016,-177.076,8.301,148.774
C00717=1149.633,289.835,-71.986,-177.078,8.298,148.774
C00718=1149.637,289.587,-71.957,-177.081,8.295,148.774
C00719=1149.642,289.339,-71.926,-177.084,8.292,148.774
C00720=1149.645,289.090,-71.896,-177.087,8.288,148.774
C00721=1149.650,288.842,-71.865,-177.089,8.284,148.774
C00722=1149.654,288.593,-71.836,-177.092,8.282,148.774
C00723=1149.658,288.346,-71.806,-177.094,8.278,148.773
C00724=1149.663,288.097,-71.776,-177.097,8.275,148.773
C00725=1149.668,287.822,-71.742,-177.100,8.272,148.773
C00726=1149.672,287.546,-71.710,-177.103,8.268,148.773
C00727=1149.677,287.272,-71.676,-177.106,8.265,148.773
C00728=1149.681,286.997,-71.643,-177.109,8.261,148.773
C00729=1149.686,286.748,-71.613,-177.112,8.258,148.773
C00730=1149.690,286.500,-71.583,-177.115,8.255,148.773
C00731=1149.694,286.252,-71.553,-177.117,8.251,148.773
C00732=1149.698,286.004,-71.524,-177.120,8.248,148.773
C00733=1149.703,285.755,-71.494,-177.122,8.245,148.773
C00734=1149.707,285.508,-71.464,-177.125,8.241,148.773
C00735=1149.711,285.260,-71.434,-177.128,8.238,148.773
C00736=1149.716,285.011,-71.405,-177.130,8.235,148.773
C00737=1149.720,284.762,-71.374,-177.133,8.232,148.773
C00738=1149.724,284.514,-71.344,-177.136,8.229,148.773
C00739=1149.728,284.266,-71.315,-177.138,8.226,148.773
C00740=1149.732,284.018,-71.285,-177.141,8.223,148.773
C00741=1149.736,283.770,-71.256,-177.143,8.220,148.773
C00742=1149.742,283.522,-71.226,-177.147,8.216,148.773
C00743=1149.746,283.274,-71.196,-177.150,8.213,148.773
C00744=1149.750,283.026,-71.166,-177.152,8.210,148.772
C00745=1149.754,282.777,-71.137,-177.155,8.207,148.772
C00746=1149.758,282.529,-71.107,-177.157,8.204,148.773
C00747=1149.762,282.281,-71.078,-177.160,8.201,148.772
C00748=1149.767,282.032,-71.048,-177.162,8.198,148.772
C00749=1149.772,281.784,-71.019,-177.165,8.194,148.772
C00750=1149.776,281.536,-70.989,-177.168,8.191,148.772
C00751=1149.780,281.288,-70.959,-177.171,8.188,148.772
C00752=1149.784,281.040,-70.929,-177.173,8.184,148.772
C00753=1149.788,280.792,-70.900,-177.176,8.182,148.772
C00754=1149.792,280.543,-70.871,-177.179,8.179,148.772
C00755=1149.796,280.295,-70.841,-177.181,8.175,148.772
C00756=1149.801,280.047,-70.812,-177.184,8.172,148.772
C00757=1149.805,279.799,-70.782,-177.187,8.169,148.772
C00758=1149.809,279.550,-70.753,-177.189,8.166,148.772
C00759=1149.814,279.303,-70.724,-177.192,8.162,148.772
C00760=1149.818,279.054,-70.694,-177.195,8.159,148.772
C00761=1149.822,278.806,-70.665,-177.197,8.156,148.772
C00762=1149.827,278.557,-70.636,-177.200,8.153,148.772
C00763=1149.831,278.309,-70.607,-177.203,8.150,148.772
C00764=1149.835,278.061,-70.577,-177.206,8.147,148.772
C00765=1149.839,277.813,-70.548,-177.208,8.144,148.772
C00766=1149.843,277.564,-70.518,-177.211,8.141,148.772
C00767=1149.848,277.317,-70.489,-177.214,8.138,148.772
C00768=1149.852,277.068,-70.460,-177.216,8.135,148.772
C00769=1149.857,276.820,-70.431,-177.219,8.131,148.772
C00770=1149.861,276.571,-70.401,-177.222,8.128,148.772
C00771=1149.865,276.323,-70.372,-177.225,8.125,148.772
C00772=1149.869,276.075,-70.343,-177.227,8.122,148.772
C00773=1149.873,275.826,-70.313,-177.230,8.119,148.772
C00774=1149.879,275.578,-70.285,-177.233,8.116,148.772
C00775=1149.882,275.330,-70.256,-177.235,8.113,148.772
C00776=1149.886,275.082,-70.226,-177.238,8.110,148.772
C00777=1149.891,274.833,-70.198,-177.241,8.107,148.772
C00778=1149.895,274.585,-70.168,-177.243,8.104,148.772
C00779=1149.900,274.337,-70.139,-177.246,8.101,148.772
C00780=1149.904,274.089,-70.110,-177.248,8.098,148.772
C00781=1149.908,273.840,-70.082,-177.252,8.094,148.772
C00782=1149.912,273.592,-70.052,-177.255,8.091,148.772
C00783=1149.916,273.343,-70.023,-177.257,8.088,148.772
C00784=1149.921,273.096,-69.994,-177.260,8.085,148.772
C00785=1149.925,272.847,-69.965,-177.262,8.082,148.772
C00786=1149.929,272.599,-69.937,-177.265,8.079,148.772
C00787=1149.933,272.351,-69.907,-177.268,8.076,148.772
C00788=1149.938,272.102,-69.879,-177.270,8.073,148.772
C00789=1149.942,271.854,-69.849,-177.273,8.070,148.772
C00790=1149.947,271.605,-69.821,-177.276,8.067,148.772
C00791=1149.951,271.358,-69.792,-177.278,8.064,148.772
C00792=1149.955,271.109,-69.763,-177.281,8.061,148.772
C00793=1149.960,270.861,-69.734,-177.284,8.058,148.772
C00794=1149.963,270.612,-69.706,-177.287,8.055,148.772
C00795=1149.968,270.365,-69.677,-177.289,8.052,148.772
C00796=1149.973,270.116,-69.648,-177.292,8.049,148.772
C00797=1149.977,269.868,-69.619,-177.294,8.046,148.772
C00798=1149.981,269.620,-69.591,-177.298,8.042,148.772
C00799=1149.985,269.371,-69.561,-177.301,8.039,148.772
C00800=1149.990,269.123,-69.533,-177.303,8.036,148.772
C00801=1149.994,268.875,-69.505,-177.306,8.033,148.772
C00802=1149.998,268.626,-69.475,-177.308,8.030,148.772
C00803=1150.002,268.378,-69.447,-177.311,8.027,148.772
C00804=1150.007,268.130,-69.419,-177.314,8.024,148.772
C00805=1150.011,267.881,-69.389,-177.317,8.021,148.772
C00806=1150.015,267.633,-69.361,-177.319,8.018,148.772
C00807=1150.020,267.385,-69.333,-177.322,8.015,148.772
C00808=1150.024,267.136,-69.303,-177.325,8.012,148.772
C00809=1150.028,266.888,-69.275,-177.327,8.009,148.772
C00810=1150.033,266.640,-69.247,-177.330,8.006,148.772
C00811=1150.037,266.391,-69.219,-177.333,8.003,148.772
C00812=1150.042,266.143,-69.190,-177.335,8.000,148.772
C00813=1150.045,265.895,-69.162,-177.338,7.997,148.772
C00814=1150.050,265.646,-69.133,-177.341,7.994,148.772
C00815=1150.055,265.398,-69.104,-177.344,7.991,148.772
C00816=1150.059,265.149,-69.076,-177.346,7.988,148.772
C00817=1150.064,264.902,-69.047,-177.349,7.985,148.772
C00818=1150.067,264.653,-69.019,-177.352,7.982,148.772
C00819=1150.072,264.405,-68.991,-177.354,7.979,148.772
C00820=1150.076,264.156,-68.963,-177.357,7.976,148.772
C00821=1150.081,263.907,-68.934,-177.360,7.973,148.772
C00822=1150.085,263.660,-68.906,-177.363,7.970,148.772
C00823=1150.090,263.411,-68.877,-177.365,7.967,148.772
C00824=1150.094,263.163,-68.849,-177.368,7.964,148.772
C00825=1150.098,262.914,-68.821,-177.371,7.961,148.772
C00826=1150.103,262.666,-68.793,-177.374,7.958,148.773
C00827=1150.106,262.417,-68.765,-177.376,7.955,148.772
C00828=1150.112,262.169,-68.736,-177.379,7.952,148.772
C00829=1150.116,261.897,-68.705,-177.382,7.948,148.772
C00830=1150.120,261.623,-68.674,-177.385,7.946,148.773
C00831=1150.125,261.349,-68.643,-177.388,7.943,148.773
C00832=1150.130,261.076,-68.612,-177.391,7.939,148.773
C00833=1150.134,260.828,-68.584,-177.394,7.936,148.773
C00834=1150.139,260.579,-68.556,-177.397,7.933,148.773
C00835=1150.143,260.331,-68.528,-177.399,7.930,148.773
C00836=1150.147,260.082,-68.500,-177.402,7.927,148.773
C00837=1150.152,259.834,-68.471,-177.405,7.924,148.773
C00838=1150.156,259.586,-68.443,-177.408,7.921,148.773
C00839=1150.160,259.337,-68.416,-177.411,7.918,148.773
C00840=1150.165,259.088,-68.387,-177.413,7.915,148.773
C00841=1150.169,258.840,-68.360,-177.416,7.912,148.773
C00842=1150.174,258.592,-68.332,-177.418,7.909,148.773
C00843=1150.177,258.344,-68.304,-177.421,7.906,148.773
C00844=1150.182,258.096,-68.275,-177.424,7.903,148.773
C00845=1150.187,257.846,-68.248,-177.426,7.901,148.773
C00846=1150.191,257.599,-68.220,-177.429,7.898,148.773
C00847=1150.195,257.350,-68.192,-177.432,7.895,148.773
C00848=1150.200,257.102,-68.164,-177.435,7.892,148.773
C00849=1150.204,256.853,-68.136,-177.437,7.889,148.773
C00850=1150.208,256.605,-68.108,-177.440,7.887,148.774
C00851=1150.212,256.357,-68.081,-177.443,7.884,148.774
C00852=1150.217,256.107,-68.053,-177.446,7.881,148.774
C00853=1150.222,255.859,-68.025,-177.448,7.878,148.774
C00854=1150.226,255.612,-67.997,-177.451,7.875,148.774
C00855=1150.230,255.362,-67.970,-177.454,7.872,148.774
C00856=1150.234,255.115,-67.942,-177.457,7.869,148.774
C00857=1150.238,254.866,-67.914,-177.459,7.866,148.774
C00858=1150.244,254.617,-67.886,-177.462,7.863,148.774
C00859=1150.248,254.369,-67.858,-177.465,7.860,148.774
C00860=1150.252,254.120,-67.831,-177.467,7.857,148.774
C00861=1150.256,253.872,-67.803,-177.470,7.854,148.774
C00862=1150.261,253.624,-67.776,-177.473,7.851,148.774
C00863=1150.265,253.375,-67.748,-177.476,7.848,148.774
C00864=1150.269,253.127,-67.720,-177.479,7.845,148.774
C00865=1150.274,252.879,-67.693,-177.481,7.842,148.774
C00866=1150.277,252.630,-67.665,-177.484,7.839,148.774
C00867=1150.283,252.381,-67.637,-177.486,7.837,148.774
C00868=1150.287,252.134,-67.609,-177.489,7.834,148.775
C00869=1150.291,251.884,-67.582,-177.492,7.831,148.775
C00870=1150.296,251.636,-67.555,-177.495,7.828,148.775
C00871=1150.300,251.388,-67.527,-177.497,7.825,148.775
C00872=1150.305,251.139,-67.500,-177.500,7.822,148.775
C00873=1150.309,250.891,-67.472,-177.503,7.820,148.775
C00874=1150.313,250.642,-67.445,-177.506,7.817,148.775
C00875=1150.318,250.394,-67.418,-177.509,7.814,148.775
C00876=1150.322,250.146,-67.390,-177.511,7.811,148.775
C00877=1150.326,249.897,-67.363,-177.514,7.808,148.775
C00878=1150.331,249.648,-67.336,-177.517,7.805,148.775
C00879=1150.335,249.400,-67.308,-177.520,7.802,148.775
C00880=1150.339,249.151,-67.280,-177.522,7.800,148.775
C00881=1150.344,248.903,-67.253,-177.525,7.797,148.775
C00882=1150.348,248.655,-67.225,-177.527,7.794,148.776
C00883=1150.352,248.407,-67.199,-177.530,7.791,148.776
C00884=1150.357,248.158,-67.172,-177.533,7.788,148.776
C00885=1150.361,247.909,-67.145,-177.536,7.785,148.776
C00886=1150.365,247.661,-67.117,-177.539,7.783,148.776
C00887=1150.370,247.413,-67.090,-177.542,7.780,148.776
C00888=1150.375,247.164,-67.063,-177.545,7.777,148.776
C00889=1150.379,246.916,-67.036,-177.547,7.774,148.776
C00890=1150.383,246.666,-67.008,-177.550,7.771,148.776
C00891=1150.388,246.419,-66.980,-177.552,7.769,148.776
C00892=1150.392,246.170,-66.953,-177.555,7.766,148.777
C00893=1150.396,245.922,-66.927,-177.558,7.763,148.777
C00894=1150.401,245.673,-66.900,-177.561,7.760,148.777
C00895=1150.406,245.425,-66.873,-177.564,7.757,148.777
C00896=1150.410,245.176,-66.845,-177.566,7.754,148.777
C00897=1150.414,244.927,-66.818,-177.569,7.751,148.777
C00898=1150.418,244.679,-66.792,-177.572,7.748,148.777
C00899=1150.423,244.431,-66.765,-177.575,7.745,148.777
C00900=1150.428,244.182,-66.738,-177.577,7.743,148.777
C00901=1150.432,243.934,-66.711,-177.580,7.740,148.777
C00902=1150.437,243.685,-66.684,-177.583,7.738,148.777
C00903=1150.440,243.436,-66.657,-177.586,7.735,148.778
C00904=1150.445,243.188,-66.630,-177.588,7.732,148.778
C00905=1150.450,242.939,-66.603,-177.591,7.729,148.778
C00906=1150.454,242.691,-66.575,-177.594,7.726,148.778
C00907=1150.458,242.442,-66.549,-177.597,7.723,148.778
C00908=1150.463,242.194,-66.522,-177.599,7.721,148.778
C00909=1150.467,241.945,-66.495,-177.602,7.718,148.778
C00910=1150.471,241.697,-66.468,-177.605,7.715,148.778
C00911=1150.476,241.449,-66.441,-177.607,7.712,148.778
C00912=1150.481,241.200,-66.414,-177.610,7.709,148.778
C00913=1150.484,240.951,-66.387,-177.613,7.707,148.779
C00914=1150.489,240.703,-66.360,-177.616,7.704,148.779
C00915=1150.494,240.454,-66.334,-177.618,7.702,148.779
C00916=1150.498,240.206,-66.308,-177.621,7.699,148.779
C00917=1150.502,239.957,-66.281,-177.624,7.696,148.779
C00918=1150.507,239.709,-66.253,-177.627,7.693,148.779
C00919=1150.511,239.460,-66.227,-177.629,7.690,148.779
C00920=1150.516,239.211,-66.201,-177.632,7.687,148.779
C00921=1150.520,238.963,-66.174,-177.636,7.684,148.779
C00922=1150.524,238.715,-66.147,-177.638,7.682,148.780
C00923=1150.529,238.466,-66.120,-177.641,7.679,148.780
C00924=1150.533,238.217,-66.094,-177.643,7.676,148.780
C00925=1150.538,237.969,-66.067,-177.646,7.673,148.780
C00926=1150.542,237.721,-66.041,-177.649,7.670,148.780
C00927=1150.547,237.472,-66.014,-177.652,7.668,148.780
C00928=1150.551,237.223,-65.988,-177.654,7.665,148.780
C00929=1150.555,236.975,-65.961,-177.657,7.663,148.780
C00930=1150.560,236.726,-65.935,-177.660,7.660,148.780
C00931=1150.564,236.478,-65.908,-177.663,7.657,148.780
C00932=1150.569,236.229,-65.881,-177.665,7.654,148.781
C00933=1150.574,235.957,-65.853,-177.668,7.651,148.781
C00934=1150.579,235.686,-65.824,-177.671,7.649,148.781
C00935=1150.583,235.414,-65.795,-177.674,7.646,148.781
C00936=1150.589,235.142,-65.766,-177.677,7.643,148.781
C00937=1150.592,234.894,-65.740,-177.680,7.640,148.781
C00938=1150.597,234.645,-65.713,-177.683,7.637,148.781
C00939=1150.601,234.397,-65.687,-177.686,7.634,148.782
C00940=1150.606,234.147,-65.661,-177.689,7.631,148.782
C00941=1150.610,233.899,-65.634,-177.691,7.629,148.782
C00942=1150.615,233.650,-65.608,-177.694,7.626,148.782
C00943=1150.619,233.402,-65.581,-177.696,7.623,148.782
C00944=1150.623,233.153,-65.556,-177.700,7.621,148.782
C00945=1150.628,232.905,-65.529,-177.702,7.618,148.782
C00946=1150.633,232.657,-65.503,-177.705,7.615,148.782
C00947=1150.637,232.408,-65.476,-177.707,7.613,148.783
C00948=1150.642,232.159,-65.450,-177.710,7.610,148.783
C00949=1150.646,231.910,-65.425,-177.713,7.607,148.783
C00950=1150.651,231.662,-65.398,-177.716,7.604,148.783
C00951=1150.655,231.413,-65.372,-177.719,7.602,148.783
C00952=1150.659,231.164,-65.346,-177.721,7.599,148.783
C00953=1150.664,230.916,-65.319,-177.724,7.596,148.783
C00954=1150.668,230.668,-65.294,-177.727,7.593,148.783
C00955=1150.673,230.419,-65.268,-177.730,7.591,148.784
C00956=1150.677,230.170,-65.241,-177.732,7.589,148.784
C00957=1150.682,229.922,-65.215,-177.735,7.586,148.784
C00958=1150.686,229.673,-65.189,-177.738,7.583,148.784
C00959=1150.690,229.424,-65.164,-177.741,7.580,148.784
C00960=1150.695,229.176,-65.137,-177.744,7.577,148.784
C00961=1150.700,228.927,-65.111,-177.746,7.575,148.784
C00962=1150.704,228.679,-65.085,-177.749,7.572,148.784
C00963=1150.708,228.430,-65.060,-177.752,7.569,148.785
C00964=1150.713,228.181,-65.033,-177.755,7.567,148.785
C00965=1150.717,227.933,-65.007,-177.757,7.565,148.785
C00966=1150.722,227.684,-64.981,-177.760,7.562,148.785
C00967=1150.726,227.436,-64.956,-177.763,7.559,148.785
C00968=1150.730,227.187,-64.930,-177.766,7.556,148.785
C00969=1150.736,226.938,-64.904,-177.768,7.554,148.786
C00970=1150.740,226.690,-64.878,-177.771,7.551,148.786
C00971=1150.744,226.441,-64.852,-177.774,7.548,148.786
C00972=1150.748,226.193,-64.826,-177.777,7.546,148.786
C00973=1150.753,225.945,-64.801,-177.779,7.544,148.786
C00974=1150.757,225.696,-64.775,-177.782,7.541,148.786
C00975=1150.762,225.447,-64.748,-177.785,7.538,148.786
C00976=1150.766,225.198,-64.723,-177.788,7.535,148.787
C00977=1150.771,224.950,-64.697,-177.790,7.533,148.787
C00978=1150.775,224.701,-64.672,-177.793,7.530,148.787
C00979=1150.780,224.452,-64.646,-177.796,7.527,148.787
C00980=1150.784,224.204,-64.620,-177.799,7.525,148.787
C00981=1150.789,223.955,-64.595,-177.801,7.523,148.787
C00982=1150.793,223.706,-64.569,-177.804,7.520,148.787
C00983=1150.797,223.458,-64.543,-177.807,7.517,148.788
C00984=1150.802,223.209,-64.518,-177.810,7.514,148.788
C00985=1150.806,222.961,-64.492,-177.812,7.512,148.788
C00986=1150.811,222.712,-64.466,-177.815,7.509,148.788
C00987=1150.816,222.463,-64.441,-177.818,7.507,148.788
C00988=1150.820,222.214,-64.415,-177.821,7.504,148.789
C00989=1150.825,221.965,-64.390,-177.823,7.502,148.789
C00990=1150.830,221.717,-64.364,-177.826,7.499,148.789
C00991=1150.834,221.468,-64.338,-177.829,7.496,148.789
C00992=1150.838,221.220,-64.313,-177.832,7.494,148.789
C00993=1150.843,220.971,-64.287,-177.834,7.491,148.789
C00994=1150.847,220.722,-64.262,-177.838,7.488,148.790
C00995=1150.852,220.474,-64.237,-177.840,7.486,148.790
C00996=1150.856,220.225,-64.211,-177.843,7.483,148.790
C00997=1150.860,219.977,-64.186,-177.846,7.481,148.790
C00998=1150.865,219.728,-64.161,-177.849,7.478,148.790
C00999=1150.869,219.479,-64.136,-177.851,7.476,148.790
C01000=1150.873,219.230,-64.110,-177.854,7.473,148.790
C01001=1150.878,218.982,-64.084,-177.857,7.470,148.791
C01002=1150.883,218.733,-64.059,-177.859,7.468,148.791
C01003=1150.888,218.485,-64.034,-177.862,7.465,148.791
C01004=1150.892,218.236,-64.008,-177.865,7.463,148.791
C01005=1150.897,217.987,-63.984,-177.867,7.461,148.791
C01006=1150.901,217.738,-63.958,-177.870,7.458,148.791
C01007=1150.905,217.490,-63.933,-177.874,7.455,148.792
C01008=1150.910,217.241,-63.908,-177.876,7.453,148.792
C01009=1150.914,216.992,-63.882,-177.879,7.450,148.792
C01010=1150.919,216.744,-63.858,-177.882,7.447,148.792
C01011=1150.923,216.495,-63.832,-177.884,7.445,148.792
C01012=1150.928,216.247,-63.806,-177.887,7.442,148.792
C01013=1150.932,215.998,-63.782,-177.890,7.440,148.793
C01014=1150.937,215.749,-63.757,-177.892,7.438,148.793
C01015=1150.941,215.500,-63.732,-177.895,7.435,148.793
C01016=1150.946,215.251,-63.706,-177.898,7.432,148.793
C01017=1150.951,215.002,-63.681,-177.900,7.430,148.793
C01018=1150.954,214.754,-63.656,-177.904,7.428,148.794
C01019=1150.959,214.505,-63.631,-177.907,7.425,148.794
C01020=1150.964,214.256,-63.606,-177.909,7.423,148.794
C01021=1150.969,214.008,-63.581,-177.912,7.420,148.794
C01022=1150.972,213.759,-63.556,-177.915,7.417,148.794
C01023=1150.977,213.510,-63.531,-177.917,7.415,148.794
C01024=1150.982,213.262,-63.506,-177.920,7.412,148.795
C01025=1150.986,213.013,-63.481,-177.923,7.409,148.795
C01026=1150.991,212.765,-63.457,-177.925,7.407,148.795
C01027=1150.995,212.516,-63.431,-177.929,7.405,148.795
C01028=1151.000,212.267,-63.406,-177.931,7.402,148.795
C01029=1151.004,212.018,-63.382,-177.934,7.400,148.796
C01030=1151.009,211.770,-63.356,-177.937,7.397,148.796
C01031=1151.014,211.520,-63.331,-177.939,7.395,148.796
C01032=1151.018,211.272,-63.307,-177.942,7.392,148.796
C01033=1151.022,211.023,-63.281,-177.945,7.390,148.796
C01034=1151.027,210.774,-63.257,-177.948,7.388,148.797
C01035=1151.032,210.526,-63.233,-177.951,7.385,148.797
C01036=1151.036,210.277,-63.207,-177.953,7.382,148.797
C01037=1151.041,210.007,-63.180,-177.957,7.379,148.797
C01038=1151.046,209.736,-63.153,-177.959,7.376,148.797
C01039=1151.051,209.466,-63.126,-177.962,7.375,148.798
C01040=1151.056,209.195,-63.100,-177.965,7.372,148.798
C01041=1151.060,208.946,-63.075,-177.968,7.369,148.798
C01042=1151.065,208.698,-63.051,-177.971,7.366,148.798
C01043=1151.069,208.449,-63.026,-177.974,7.365,148.799
C01044=1151.074,208.200,-63.002,-177.976,7.362,148.799
C01045=1151.078,207.951,-62.976,-177.979,7.360,148.799
C01046=1151.083,207.702,-62.952,-177.982,7.357,148.799
C01047=1151.088,207.454,-62.927,-177.985,7.354,148.799
C01048=1151.092,207.205,-62.902,-177.987,7.352,148.800
C01049=1151.096,206.956,-62.878,-177.990,7.349,148.800
C01050=1151.102,206.708,-62.853,-177.993,7.348,148.800
C01051=1151.105,206.459,-62.829,-177.996,7.345,148.800
C01052=1151.111,206.210,-62.804,-177.999,7.342,148.800
C01053=1151.115,205.961,-62.780,-178.001,7.340,148.801
C01054=1151.119,205.712,-62.756,-178.004,7.337,148.801
C01055=1151.124,205.464,-62.731,-178.007,7.335,148.801
C01056=1151.128,205.215,-62.707,-178.009,7.332,148.801
C01057=1151.133,204.966,-62.682,-178.013,7.330,148.801
C01058=1151.137,204.717,-62.658,-178.015,7.328,148.802
C01059=1151.142,204.469,-62.633,-178.018,7.325,148.802
C01060=1151.147,204.220,-62.609,-178.020,7.323,148.802
C01061=1151.151,203.971,-62.584,-178.024,7.321,148.802
C01062=1151.156,203.722,-62.560,-178.026,7.318,148.802
C01063=1151.160,203.474,-62.536,-178.029,7.315,148.803
C01064=1151.165,203.225,-62.511,-178.032,7.313,148.803
C01065=1151.169,202.976,-62.487,-178.034,7.311,148.803
C01066=1151.173,202.728,-62.463,-178.037,7.308,148.803
C01067=1151.179,202.478,-62.439,-178.040,7.306,148.803
C01068=1151.183,202.230,-62.415,-178.043,7.304,148.804
C01069=1151.188,201.981,-62.390,-178.045,7.301,148.804
C01070=1151.192,201.732,-62.366,-178.048,7.299,148.804
C01071=1151.196,201.484,-62.341,-178.051,7.296,148.804
C01072=1151.201,201.235,-62.317,-178.054,7.294,148.805
C01073=1151.206,200.985,-62.293,-178.057,7.291,148.805
C01074=1151.210,200.737,-62.269,-178.059,7.290,148.805
C01075=1151.215,200.488,-62.245,-178.062,7.287,148.805
C01076=1151.220,200.240,-62.220,-178.065,7.285,148.806
C01077=1151.224,199.991,-62.196,-178.068,7.282,148.806
C01078=1151.228,199.742,-62.172,-178.070,7.280,148.806
C01079=1151.233,199.493,-62.148,-178.073,7.277,148.806
C01080=1151.238,199.244,-62.124,-178.076,7.276,148.807
C01081=1151.242,198.995,-62.100,-178.078,7.273,148.807
C01082=1151.247,198.747,-62.076,-178.082,7.270,148.807
C01083=1151.251,198.498,-62.052,-178.084,7.268,148.807
C01084=1151.256,198.248,-62.028,-178.087,7.265,148.807
C01085=1151.260,198.000,-62.004,-178.089,7.263,148.808
C01086=1151.265,197.752,-61.980,-178.093,7.261,148.808
C01087=1151.269,197.503,-61.956,-178.095,7.259,148.808
C01088=1151.274,197.254,-61.932,-178.098,7.256,148.808
C01089=1151.279,197.006,-61.908,-178.100,7.254,148.808
C01090=1151.283,196.756,-61.884,-178.104,7.251,148.809
C01091=1151.287,196.507,-61.860,-178.106,7.249,148.809
C01092=1151.292,196.258,-61.836,-178.109,7.247,148.809
C01093=1151.297,196.010,-61.812,-178.112,7.245,148.810
C01094=1151.301,195.761,-61.789,-178.115,7.242,148.810
C01095=1151.306,195.512,-61.765,-178.117,7.240,148.810
C01096=1151.311,195.263,-61.741,-178.120,7.237,148.810
C01097=1151.316,195.015,-61.717,-178.123,7.236,148.811
C01098=1151.320,194.766,-61.694,-178.126,7.233,148.811
C01099=1151.325,194.517,-61.669,-178.128,7.231,148.811
C01100=1151.329,194.268,-61.646,-178.131,7.228,148.811
C01101=1151.333,194.019,-61.622,-178.134,7.226,148.811
C01102=1151.338,193.770,-61.598,-178.137,7.223,148.812
C01103=1151.342,193.522,-61.574,-178.139,7.222,148.812
C01104=1151.347,193.273,-61.551,-178.143,7.219,148.812
C01105=1151.352,193.024,-61.528,-178.145,7.217,148.812
C01106=1151.356,192.775,-61.503,-178.148,7.214,148.813
C01107=1151.361,192.526,-61.480,-178.150,7.212,148.813
C01108=1151.365,192.278,-61.456,-178.153,7.210,148.813
C01109=1151.370,192.029,-61.433,-178.156,7.208,148.813
C01110=1151.374,191.780,-61.409,-178.159,7.205,148.814
C01111=1151.379,191.531,-61.385,-178.162,7.203,148.814
C01112=1151.384,191.282,-61.362,-178.164,7.200,148.814
C01113=1151.388,191.033,-61.339,-178.167,7.199,148.814
C01114=1151.393,190.785,-61.314,-178.170,7.196,148.815
C01115=1151.397,190.536,-61.291,-178.173,7.194,148.815
C01116=1151.402,190.287,-61.268,-178.175,7.191,148.815
C01117=1151.407,190.038,-61.244,-178.178,7.189,148.815
C01118=1151.411,189.789,-61.220,-178.181,7.187,148.816
C01119=1151.416,189.540,-61.197,-178.184,7.185,148.816
C01120=1151.421,189.291,-61.174,-178.186,7.183,148.816
C01121=1151.425,189.042,-61.150,-178.189,7.180,148.816
C01122=1151.430,188.793,-61.127,-178.192,7.178,148.817
C01123=1151.434,188.545,-61.103,-178.195,7.176,148.817
C01124=1151.439,188.296,-61.079,-178.197,7.174,148.817
C01125=1151.444,188.047,-61.056,-178.201,7.171,148.818
C01126=1151.448,187.798,-61.033,-178.203,7.169,148.818
C01127=1151.452,187.549,-61.010,-178.206,7.166,148.818
C01128=1151.458,187.301,-60.987,-178.209,7.165,148.818
C01129=1151.462,187.052,-60.964,-178.212,7.162,148.818
C01130=1151.467,186.803,-60.940,-178.214,7.160,148.819
C01131=1151.472,186.554,-60.916,-178.216,7.158,148.819
C01132=1151.476,186.305,-60.893,-178.220,7.155,148.819
C01133=1151.480,186.056,-60.870,-178.222,7.154,148.820
C01134=1151.485,185.807,-60.847,-178.225,7.151,148.820
C01135=1151.490,185.558,-60.823,-178.228,7.149,148.820
C01136=1151.494,185.309,-60.800,-178.231,7.146,148.821
C01137=1151.499,185.060,-60.777,-178.233,7.144,148.821
C01138=1151.503,184.812,-60.754,-178.237,7.142,148.821
C01139=1151.508,184.563,-60.731,-178.239,7.140,148.821
C01140=1151.513,184.314,-60.707,-178.242,7.138,148.821
C01141=1151.518,184.044,-60.682,-178.245,7.135,148.822
C01142=1151.523,183.775,-60.658,-178.248,7.133,148.822
C01143=1151.528,183.504,-60.633,-178.251,7.131,148.823
C01144=1151.533,183.235,-60.607,-178.254,7.128,148.823
C01145=1151.537,182.987,-60.585,-178.257,7.126,148.823
C01146=1151.542,182.738,-60.562,-178.260,7.124,148.823
C01147=1151.547,182.489,-60.538,-178.262,7.122,148.823
C01148=1151.552,182.240,-60.515,-178.265,7.119,148.824
C01149=1151.555,181.991,-60.492,-178.268,7.117,148.824
C01150=1151.560,181.742,-60.469,-178.271,7.115,148.824
C01151=1151.565,181.494,-60.446,-178.273,7.113,148.825
C01152=1151.570,181.244,-60.424,-178.276,7.111,148.825
C01153=1151.574,180.995,-60.401,-178.279,7.108,148.825
C01154=1151.579,180.746,-60.377,-178.281,7.106,148.826
C01155=1151.583,180.497,-60.354,-178.285,7.104,148.826
C01156=1151.588,180.249,-60.331,-178.287,7.102,148.826
C01157=1151.593,180.000,-60.309,-178.290,7.100,148.826
C01158=1151.597,179.751,-60.286,-178.293,7.097,148.827
C01159=1151.602,179.502,-60.263,-178.295,7.095,148.827
C01160=1151.606,179.253,-60.240,-178.298,7.093,148.827
C01161=1151.612,179.004,-60.218,-178.301,7.091,148.828
C01162=1151.616,178.755,-60.195,-178.303,7.089,148.828
C01163=1151.620,178.506,-60.172,-178.307,7.086,148.828
C01164=1151.625,178.257,-60.149,-178.309,7.085,148.828
C01165=1151.630,178.009,-60.126,-178.311,7.083,148.829
C01166=1151.635,177.760,-60.103,-178.315,7.080,148.829
C01167=1151.639,177.510,-60.081,-178.317,7.078,148.829
C01168=1151.644,177.261,-60.058,-178.321,7.076,148.830
C01169=1151.648,177.013,-60.035,-178.323,7.074,148.830
C01170=1151.653,176.763,-60.013,-178.326,7.072,148.830
C01171=1151.657,176.515,-59.990,-178.329,7.069,148.830
C01172=1151.663,176.266,-59.968,-178.331,7.067,148.831
C01173=1151.667,176.017,-59.945,-178.334,7.066,148.831
C01174=1151.671,175.768,-59.922,-178.337,7.063,148.831
C01175=1151.676,175.519,-59.899,-178.339,7.061,148.831
C01176=1151.681,175.270,-59.876,-178.343,7.058,148.832
C01177=1151.685,175.021,-59.854,-178.345,7.057,148.832
C01178=1151.689,174.772,-59.832,-178.348,7.055,148.833
C01179=1151.695,174.523,-59.809,-178.351,7.052,148.833
C01180=1151.699,174.275,-59.787,-178.354,7.050,148.833
C01181=1151.704,174.025,-59.764,-178.356,7.048,148.833
C01182=1151.708,173.777,-59.742,-178.359,7.046,148.834
C01183=1151.713,173.527,-59.719,-178.362,7.044,148.834
C01184=1151.718,173.278,-59.697,-178.364,7.042,148.834
C01185=1151.722,173.030,-59.674,-178.368,7.040,148.835
C01186=1151.727,172.780,-59.652,-178.370,7.037,148.835
C01187=1151.732,172.532,-59.629,-178.373,7.036,148.835
C01188=1151.737,172.283,-59.607,-178.376,7.033,148.835
C01189=1151.741,172.033,-59.585,-178.379,7.031,148.836
C01190=1151.746,171.785,-59.562,-178.381,7.029,148.836
C01191=1151.751,171.536,-59.540,-178.384,7.027,148.836
C01192=1151.755,171.288,-59.517,-178.387,7.025,148.837
C01193=1151.759,171.038,-59.495,-178.389,7.023,148.837
C01194=1151.764,170.789,-59.473,-178.392,7.020,148.837
C01195=1151.769,170.540,-59.451,-178.395,7.019,148.838
C01196=1151.773,170.291,-59.428,-178.398,7.017,148.838
C01197=1151.779,170.042,-59.406,-178.401,7.014,148.838
C01198=1151.783,169.793,-59.384,-178.404,7.013,148.839
C01199=1151.787,169.544,-59.361,-178.406,7.011,148.839
C01200=1151.792,169.296,-59.339,-178.409,7.009,148.839
C01201=1151.797,169.046,-59.317,-178.412,7.006,148.840
C01202=1151.802,168.797,-59.295,-178.415,7.005,148.840
C01203=1151.806,168.549,-59.272,-178.417,7.002,148.840
C01204=1151.811,168.300,-59.251,-178.420,7.000,148.840
C01205=1151.816,168.050,-59.228,-178.423,6.998,148.841
C01206=1151.820,167.802,-59.206,-178.425,6.996,148.841
C01207=1151.825,167.552,-59.184,-178.428,6.994,148.841
C01208=1151.830,167.304,-59.163,-178.431,6.992,148.842
C01209=1151.834,167.055,-59.139,-178.434,6.990,148.842
C01210=1151.839,166.806,-59.118,-178.436,6.988,148.842
C01211=1151.843,166.557,-59.095,-178.440,6.986,148.843
C01212=1151.848,166.308,-59.074,-178.442,6.984,148.843
C01213=1151.853,166.059,-59.052,-178.445,6.982,148.843
C01214=1151.858,165.810,-59.029,-178.448,6.979,148.844
C01215=1151.862,165.560,-59.007,-178.451,6.978,148.844
C01216=1151.867,165.312,-58.986,-178.453,6.976,148.844
C01217=1151.872,165.062,-58.964,-178.455,6.974,148.845
C01218=1151.876,164.814,-58.942,-178.459,6.971,148.845
C01219=1151.881,164.564,-58.920,-178.461,6.970,148.845
C01220=1151.886,164.316,-58.898,-178.464,6.968,148.846
C01221=1151.890,164.066,-58.876,-178.467,6.965,148.846
C01222=1151.895,163.817,-58.854,-178.470,6.963,148.846
C01223=1151.900,163.568,-58.832,-178.472,6.961,148.846
C01224=1151.905,163.319,-58.810,-178.475,6.960,148.847
C01225=1151.909,163.070,-58.788,-178.478,6.957,148.847
C01226=1151.914,162.821,-58.766,-178.481,6.955,148.848
C01227=1151.919,162.573,-58.745,-178.483,6.953,148.848
C01228=1151.923,162.324,-58.723,-178.486,6.952,148.848
C01229=1151.928,162.075,-58.701,-178.489,6.949,148.848
C01230=1151.932,161.826,-58.679,-178.492,6.947,148.849
C01231=1151.937,161.577,-58.657,-178.495,6.946,148.849
C01232=1151.942,161.328,-58.636,-178.497,6.944,148.850
C01233=1151.946,161.078,-58.614,-178.500,6.941,148.850
C01234=1151.951,160.830,-58.593,-178.503,6.939,148.850
C01235=1151.955,160.580,-58.571,-178.506,6.938,148.850
C01236=1151.960,160.332,-58.549,-178.508,6.936,148.851
C01237=1151.965,160.083,-58.527,-178.512,6.933,148.851
C01238=1151.970,159.834,-58.505,-178.514,6.932,148.852
C01239=1151.975,159.584,-58.484,-178.516,6.929,148.852
C01240=1151.979,159.335,-58.462,-178.519,6.928,148.852
C01241=1151.984,159.086,-58.440,-178.522,6.925,148.852
C01242=1151.989,158.838,-58.419,-178.525,6.923,148.853
C01243=1151.993,158.588,-58.397,-178.528,6.922,148.853
C01244=1151.998,158.339,-58.376,-178.531,6.920,148.854
C01245=1152.003,158.070,-58.353,-178.534,6.917,148.854
C01246=1152.008,157.801,-58.329,-178.537,6.916,148.854
C01247=1152.013,157.532,-58.306,-178.540,6.913,148.855
C01248=1152.018,157.263,-58.283,-178.543,6.911,148.855
C01249=1152.023,157.014,-58.261,-178.545,6.910,148.855
C01250=1152.027,156.766,-58.240,-178.548,6.907,148.856
C01251=1152.032,156.516,-58.219,-178.551,6.905,148.856
C01252=1152.037,156.267,-58.197,-178.553,6.903,148.856
C01253=1152.042,156.019,-58.175,-178.556,6.902,148.857
C01254=1152.047,155.770,-58.154,-178.559,6.900,148.857
C01255=1152.051,155.520,-58.132,-178.562,6.897,148.857
C01256=1152.056,155.271,-58.111,-178.565,6.896,148.858
C01257=1152.060,155.023,-58.090,-178.568,6.894,148.858
C01258=1152.065,154.773,-58.069,-178.570,6.892,148.858
C01259=1152.070,154.524,-58.047,-178.572,6.890,148.859
C01260=1152.075,154.275,-58.026,-178.576,6.888,148.859
C01261=1152.080,154.026,-58.005,-178.578,6.886,148.860
C01262=1152.083,153.777,-57.983,-178.581,6.884,148.860
C01263=1152.089,153.528,-57.962,-178.584,6.882,148.860
C01264=1152.093,153.279,-57.941,-178.587,6.881,148.861
C01265=1152.099,153.030,-57.920,-178.590,6.878,148.861
C01266=1152.103,152.782,-57.898,-178.593,6.876,148.861
C01267=1152.107,152.532,-57.877,-178.595,6.874,148.862
C01268=1152.112,152.282,-57.856,-178.598,6.873,148.862
C01269=1152.117,152.034,-57.835,-178.600,6.871,148.862
C01270=1152.122,151.785,-57.814,-178.603,6.869,148.863
C01271=1152.126,151.535,-57.792,-178.606,6.867,148.863
C01272=1152.131,151.286,-57.771,-178.609,6.865,148.863
C01273=1152.136,151.038,-57.749,-178.612,6.863,148.864
C01274=1152.141,150.789,-57.729,-178.614,6.861,148.864
C01275=1152.146,150.539,-57.708,-178.617,6.860,148.865
C01276=1152.151,150.291,-57.686,-178.620,6.858,148.865
C01277=1152.154,150.041,-57.666,-178.623,6.855,148.865
C01278=1152.160,149.792,-57.645,-178.625,6.853,148.866
C01279=1152.164,149.543,-57.623,-178.628,6.852,148.866
C01280=1152.169,149.294,-57.603,-178.631,6.850,148.866
C01281=1152.174,149.045,-57.582,-178.633,6.848,148.867
C01282=1152.179,148.796,-57.561,-178.636,6.846,148.867
C01283=1152.183,148.547,-57.539,-178.639,6.844,148.867
C01284=1152.188,148.297,-57.518,-178.642,6.842,148.868
C01285=1152.192,148.048,-57.498,-178.645,6.841,148.868
C01286=1152.197,147.800,-57.476,-178.648,6.839,148.869
C01287=1152.202,147.551,-57.455,-178.650,6.837,148.869
C01288=1152.207,147.302,-57.435,-178.653,6.835,148.869
C01289=1152.212,147.052,-57.414,-178.656,6.834,148.870
C01290=1152.216,146.803,-57.394,-178.659,6.831,148.870
C01291=1152.221,146.554,-57.372,-178.662,6.829,148.870
C01292=1152.225,146.305,-57.351,-178.664,6.828,148.871
C01293=1152.230,146.056,-57.330,-178.667,6.826,148.871
C01294=1152.236,145.807,-57.309,-178.669,6.824,148.871
C01295=1152.240,145.558,-57.289,-178.672,6.822,148.872
C01296=1152.245,145.308,-57.268,-178.675,6.820,148.872
C01297=1152.250,145.059,-57.248,-178.678,6.818,148.873
C01298=1152.254,144.811,-57.226,-178.681,6.816,148.873
C01299=1152.259,144.562,-57.205,-178.683,6.814,148.873
C01300=1152.264,144.313,-57.184,-178.686,6.813,148.874
C01301=1152.268,144.064,-57.164,-178.689,6.811,148.874
C01302=1152.273,143.815,-57.144,-178.692,6.809,148.874
C01303=1152.278,143.565,-57.123,-178.694,6.808,148.875
C01304=1152.282,143.316,-57.102,-178.697,6.806,148.875
C01305=1152.287,143.066,-57.081,-178.700,6.804,148.876
C01306=1152.292,142.818,-57.061,-178.703,6.802,148.876
C01307=1152.297,142.568,-57.040,-178.706,6.800,148.876
C01308=1152.301,142.319,-57.019,-178.708,6.798,148.877
C01309=1152.306,142.070,-56.998,-178.711,6.796,148.877
C01310=1152.311,141.821,-56.978,-178.714,6.795,148.878
C01311=1152.315,141.572,-56.958,-178.716,6.793,148.878
C01312=1152.320,141.323,-56.937,-178.719,6.791,148.878
C01313=1152.325,141.074,-56.916,-178.722,6.790,148.879
C01314=1152.329,140.825,-56.896,-178.725,6.788,148.879
C01315=1152.334,140.576,-56.875,-178.727,6.786,148.880
C01316=1152.339,140.326,-56.855,-178.731,6.784,148.880
C01317=1152.344,140.077,-56.834,-178.733,6.782,148.880
C01318=1152.349,139.828,-56.814,-178.736,6.780,148.881
C01319=1152.353,139.579,-56.794,-178.739,6.778,148.881
C01320=1152.358,139.330,-56.773,-178.741,6.777,148.881
C01321=1152.363,139.081,-56.752,-178.744,6.775,148.882
C01322=1152.368,138.833,-56.732,-178.747,6.773,148.882
C01323=1152.373,138.583,-56.712,-178.750,6.772,148.883
C01324=1152.378,138.334,-56.692,-178.752,6.770,148.883
C01325=1152.382,138.085,-56.671,-178.755,6.768,148.883
C01326=1152.387,137.836,-56.651,-178.758,6.766,148.884
C01327=1152.392,137.587,-56.630,-178.760,6.765,148.884
C01328=1152.397,137.337,-56.610,-178.763,6.763,148.885
C01329=1152.401,137.088,-56.590,-178.766,6.760,148.885
C01330=1152.406,136.839,-56.569,-178.769,6.759,148.885
C01331=1152.411,136.590,-56.549,-178.772,6.757,148.886
C01332=1152.415,136.340,-56.529,-178.775,6.755,148.886
C01333=1152.420,136.091,-56.509,-178.777,6.754,148.886
C01334=1152.424,135.842,-56.488,-178.780,6.752,148.887
C01335=1152.430,135.593,-56.468,-178.783,6.750,148.887
C01336=1152.435,135.344,-56.448,-178.785,6.748,148.888
C01337=1152.439,135.095,-56.428,-178.788,6.747,148.888
C01338=1152.444,134.846,-56.408,-178.791,6.745,148.888
C01339=1152.449,134.596,-56.387,-178.794,6.743,148.889
C01340=1152.454,134.348,-56.367,-178.796,6.742,148.889
C01341=1152.458,134.098,-56.347,-178.799,6.740,148.890
C01342=1152.463,133.849,-56.327,-178.802,6.738,148.890
C01343=1152.468,133.601,-56.306,-178.804,6.736,148.890
C01344=1152.473,133.351,-56.287,-178.807,6.735,148.891
C01345=1152.478,133.102,-56.266,-178.810,6.733,148.891
C01346=1152.482,132.852,-56.246,-178.813,6.731,148.892
C01347=1152.487,132.603,-56.226,-178.815,6.730,148.892
C01348=1152.492,132.354,-56.206,-178.818,6.728,148.892
C01349=1152.496,132.086,-56.184,-178.821,6.725,148.893
C01350=1152.502,131.818,-56.163,-178.824,6.724,148.893
C01351=1152.507,131.549,-56.142,-178.827,6.722,148.894
C01352=1152.513,131.281,-56.120,-178.830,6.721,148.894
C01353=1152.517,131.031,-56.100,-178.833,6.718,148.895
C01354=1152.522,130.782,-56.080,-178.836,6.716,148.895
C01355=1152.527,130.533,-56.060,-178.839,6.715,148.895
C01356=1152.531,130.284,-56.040,-178.841,6.713,148.896
C01357=1152.536,130.035,-56.020,-178.844,6.711,148.896
C01358=1152.541,129.785,-56.001,-178.847,6.709,148.897
C01359=1152.546,129.536,-55.980,-178.850,6.708,148.897
C01360=1152.550,129.287,-55.961,-178.852,6.706,148.897
C01361=1152.555,129.038,-55.941,-178.855,6.704,148.898
C01362=1152.560,128.789,-55.921,-178.858,6.703,148.898
C01363=1152.565,128.539,-55.901,-178.860,6.701,148.898
C01364=1152.569,128.290,-55.881,-178.864,6.700,148.899
C01365=1152.575,128.041,-55.862,-178.866,6.698,148.900
C01366=1152.579,127.792,-55.842,-178.869,6.696,148.900
C01367=1152.584,127.543,-55.822,-178.872,6.694,148.900
C01368=1152.589,127.293,-55.802,-178.874,6.693,148.901
C01369=1152.594,127.044,-55.783,-178.877,6.691,148.901
C01370=1152.598,126.796,-55.762,-178.880,6.689,148.901
C01371=1152.603,126.546,-55.743,-178.883,6.688,148.902
C01372=1152.608,126.297,-55.723,-178.885,6.686,148.902
C01373=1152.613,126.048,-55.704,-178.888,6.684,148.903
C01374=1152.618,125.799,-55.683,-178.891,6.682,148.903
C01375=1152.622,125.549,-55.664,-178.893,6.682,148.903
C01376=1152.628,125.300,-55.644,-178.896,6.680,148.904
C01377=1152.632,125.051,-55.625,-178.899,6.678,148.905
C01378=1152.636,124.802,-55.605,-178.901,6.677,148.905
C01379=1152.642,124.553,-55.586,-178.904,6.675,148.905
C01380=1152.646,124.303,-55.566,-178.907,6.673,148.906
C01381=1152.651,124.054,-55.546,-178.910,6.672,148.906
C01382=1152.656,123.805,-55.527,-178.912,6.670,148.907
C01383=1152.661,123.555,-55.507,-178.915,6.668,148.907
C01384=1152.666,123.307,-55.487,-178.918,6.667,148.907
C01385=1152.670,123.058,-55.468,-178.920,6.665,148.908
C01386=1152.675,122.808,-55.449,-178.923,6.663,148.908
C01387=1152.680,122.559,-55.429,-178.926,6.661,148.909
C01388=1152.685,122.310,-55.410,-178.929,6.660,148.909
C01389=1152.690,122.060,-55.390,-178.932,6.658,148.910
C01390=1152.694,121.812,-55.371,-178.935,6.657,148.910
C01391=1152.699,121.562,-55.352,-178.937,6.655,148.910
C01392=1152.704,121.313,-55.332,-178.940,6.653,148.911
C01393=1152.709,121.064,-55.313,-178.943,6.652,148.911
C01394=1152.714,120.814,-55.293,-178.945,6.650,148.912
C01395=1152.718,120.565,-55.274,-178.948,6.648,148.912
C01396=1152.723,120.316,-55.255,-178.951,6.646,148.912
C01397=1152.728,120.067,-55.235,-178.954,6.645,148.913
C01398=1152.733,119.818,-55.216,-178.956,6.644,148.913
C01399=1152.737,119.568,-55.197,-178.959,6.642,148.914
C01400=1152.743,119.320,-55.177,-178.962,6.641,148.914
C01401=1152.747,119.070,-55.158,-178.964,6.639,148.915
C01402=1152.752,118.820,-55.138,-178.967,6.637,148.915
C01403=1152.757,118.572,-55.119,-178.970,6.636,148.915
C01404=1152.762,118.322,-55.100,-178.973,6.634,148.916
C01405=1152.767,118.073,-55.080,-178.976,6.633,148.916
C01406=1152.771,117.824,-55.061,-178.978,6.631,148.917
C01407=1152.776,117.575,-55.042,-178.981,6.629,148.917
C01408=1152.781,117.326,-55.022,-178.984,6.627,148.918
C01409=1152.786,117.077,-55.004,-178.987,6.626,148.918
C01410=1152.791,116.827,-54.985,-178.989,6.624,148.918
C01411=1152.796,116.578,-54.966,-178.991,6.623,148.919
C01412=1152.800,116.329,-54.946,-178.994,6.621,148.919
C01413=1152.805,116.080,-54.927,-178.997,6.620,148.920
C01414=1152.810,115.830,-54.907,-179.000,6.618,148.920
C01415=1152.815,115.582,-54.889,-179.003,6.617,148.921
C01416=1152.820,115.332,-54.870,-179.006,6.615,148.921
C01417=1152.824,115.083,-54.851,-179.008,6.613,148.921
C01418=1152.829,114.834,-54.832,-179.011,6.612,148.922
C01419=1152.834,114.585,-54.812,-179.014,6.610,148.922
C01420=1152.839,114.335,-54.794,-179.017,6.609,148.923
C01421=1152.844,114.086,-54.775,-179.020,6.607,148.923
C01422=1152.848,113.837,-54.756,-179.022,6.606,148.924
C01423=1152.853,113.588,-54.736,-179.024,6.604,148.924
C01424=1152.858,113.338,-54.717,-179.027,6.603,148.925
C01425=1152.863,113.089,-54.699,-179.030,6.601,148.925
C01426=1152.868,112.840,-54.679,-179.033,6.600,148.926
C01427=1152.873,112.590,-54.661,-179.036,6.598,148.926
C01428=1152.878,112.342,-54.642,-179.039,6.596,148.926
C01429=1152.882,112.092,-54.623,-179.041,6.594,148.927
C01430=1152.888,111.843,-54.604,-179.043,6.594,148.927
C01431=1152.892,111.593,-54.585,-179.046,6.592,148.928
C01432=1152.897,111.345,-54.566,-179.049,6.591,148.928
C01433=1152.901,111.095,-54.547,-179.052,6.589,148.929
C01434=1152.907,110.846,-54.528,-179.055,6.587,148.929
C01435=1152.912,110.597,-54.510,-179.058,6.585,148.929
C01436=1152.916,110.347,-54.490,-179.060,6.584,148.930
C01437=1152.921,110.098,-54.472,-179.063,6.582,148.930
C01438=1152.926,109.848,-54.453,-179.066,6.582,148.931
C01439=1152.931,109.600,-54.434,-179.068,6.580,148.931
C01440=1152.936,109.351,-54.416,-179.071,6.578,148.932
C01441=1152.940,109.101,-54.396,-179.074,6.576,148.932
C01442=1152.945,108.852,-54.378,-179.076,6.575,148.933
C01443=1152.951,108.603,-54.359,-179.079,6.573,148.933
C01444=1152.955,108.353,-54.341,-179.082,6.572,148.934
C01445=1152.959,108.105,-54.322,-179.085,6.571,148.934
C01446=1152.964,107.854,-54.303,-179.087,6.569,148.934
C01447=1152.969,107.606,-54.284,-179.090,6.567,148.935
C01448=1152.975,107.356,-54.266,-179.093,6.566,148.935
C01449=1152.979,107.107,-54.248,-179.096,6.564,148.936
C01450=1152.984,106.858,-54.229,-179.099,6.563,148.936
C01451=1152.989,106.608,-54.210,-179.101,6.561,148.937
C01452=1152.993,106.359,-54.191,-179.104,6.560,148.937
C01453=1152.999,106.091,-54.171,-179.106,6.558,148.938
C01454=1153.004,105.822,-54.152,-179.109,6.557,148.938
C01455=1153.010,105.554,-54.131,-179.112,6.555,148.939
C01456=1153.015,105.286,-54.112,-179.116,6.553,148.939
C01457=1153.019,105.036,-54.093,-179.118,6.552,148.940
C01458=1153.025,104.787,-54.075,-179.121,6.551,148.940
C01459=1153.029,104.538,-54.056,-179.124,6.549,148.940
C01460=1153.034,104.288,-54.038,-179.126,6.547,148.941
C01461=1153.039,104.039,-54.019,-179.129,6.546,148.941
C01462=1153.044,103.790,-54.000,-179.132,6.545,148.942
C01463=1153.049,103.541,-53.982,-179.134,6.543,148.942
C01464=1153.053,103.291,-53.964,-179.137,6.542,148.943
C01465=1153.059,103.042,-53.945,-179.140,6.540,148.943
C01466=1153.063,102.793,-53.927,-179.143,6.539,148.944
C01467=1153.068,102.544,-53.909,-179.146,6.537,148.944
C01468=1153.073,102.294,-53.891,-179.148,6.536,148.945
C01469=1153.077,102.046,-53.872,-179.151,6.534,148.945
C01470=1153.083,101.796,-53.853,-179.154,6.533,148.946
C01471=1153.088,101.547,-53.835,-179.157,6.531,148.946
C01472=1153.092,101.297,-53.817,-179.159,6.530,148.946
C01473=1153.097,101.048,-53.799,-179.161,6.529,148.947
C01474=1153.103,100.798,-53.780,-179.164,6.527,148.947
C01475=1153.107,100.550,-53.762,-179.167,6.526,148.948
C01476=1153.112,100.300,-53.743,-179.170,6.524,148.948
C01477=1153.117,100.051,-53.725,-179.173,6.522,148.949
C01478=1153.121,99.802,-53.707,-179.175,6.521,148.949
C01479=1153.126,99.552,-53.689,-179.178,6.520,148.950
C01480=1153.131,99.303,-53.671,-179.181,6.518,148.950
C01481=1153.136,99.053,-53.652,-179.184,6.517,148.951
C01482=1153.141,98.804,-53.635,-179.186,6.516,148.951
C01483=1153.146,98.555,-53.616,-179.188,6.514,148.952
C01484=1153.151,98.306,-53.598,-179.192,6.513,148.952
C01485=1153.156,98.057,-53.580,-179.194,6.511,148.953
C01486=1153.161,97.808,-53.562,-179.197,6.509,148.953
C01487=1153.165,97.558,-53.544,-179.199,6.509,148.953
C01488=1153.170,97.309,-53.526,-179.202,6.507,148.954
C01489=1153.175,97.060,-53.508,-179.205,6.506,148.954
C01490=1153.180,96.810,-53.489,-179.208,6.504,148.955
C01491=1153.185,96.561,-53.471,-179.210,6.503,148.955
C01492=1153.190,96.312,-53.453,-179.213,6.502,148.956
C01493=1153.195,96.063,-53.435,-179.216,6.500,148.956
C01494=1153.199,95.813,-53.417,-179.219,6.498,148.957
C01495=1153.204,95.564,-53.399,-179.221,6.497,148.957
C01496=1153.209,95.314,-53.381,-179.224,6.496,148.958
C01497=1153.214,95.065,-53.363,-179.227,6.494,148.958
C01498=1153.219,94.815,-53.346,-179.230,6.493,148.959
C01499=1153.224,94.566,-53.328,-179.232,6.491,148.959
C01500=1153.229,94.317,-53.310,-179.235,6.491,148.960
C01501=1153.234,94.068,-53.292,-179.238,6.489,148.960
C01502=1153.239,93.819,-53.274,-179.240,6.487,148.961
C01503=1153.244,93.570,-53.256,-179.243,6.486,148.961
C01504=1153.248,93.320,-53.237,-179.246,6.485,148.962
C01505=1153.253,93.070,-53.219,-179.248,6.483,148.962
C01506=1153.258,92.821,-53.202,-179.251,6.482,148.962
C01507=1153.263,92.572,-53.184,-179.253,6.481,148.963
C01508=1153.268,92.322,-53.166,-179.257,6.479,148.964
C01509=1153.273,92.073,-53.148,-179.259,6.478,148.964
C01510=1153.277,91.824,-53.131,-179.262,6.476,148.964
C01511=1153.282,91.575,-53.113,-179.265,6.475,148.965
C01512=1153.287,91.325,-53.095,-179.267,6.474,148.965
C01513=1153.292,91.076,-53.077,-179.270,6.472,148.966
C01514=1153.297,90.827,-53.059,-179.273,6.470,148.966
C01515=1153.302,90.578,-53.042,-179.275,6.470,148.967
C01516=1153.307,90.328,-53.024,-179.278,6.468,148.967
C01517=1153.312,90.079,-53.006,-179.281,6.467,148.968
C01518=1153.317,89.830,-52.988,-179.283,6.466,148.968
C01519=1153.322,89.580,-52.972,-179.286,6.464,148.969
C01520=1153.327,89.331,-52.954,-179.289,6.463,148.969
C01521=1153.331,89.082,-52.936,-179.292,6.461,148.970
C01522=1153.337,88.832,-52.918,-179.294,6.460,148.970
C01523=1153.342,88.583,-52.900,-179.297,6.459,148.971
C01524=1153.347,88.334,-52.882,-179.300,6.457,148.971
C01525=1153.352,88.084,-52.865,-179.302,6.456,148.972
C01526=1153.356,87.835,-52.848,-179.305,6.455,148.972
C01527=1153.361,87.586,-52.830,-179.308,6.453,148.973
C01528=1153.366,87.336,-52.813,-179.311,6.452,148.973
C01529=1153.371,87.087,-52.795,-179.313,6.451,148.974
C01530=1153.376,86.837,-52.777,-179.316,6.449,148.974
C01531=1153.380,86.588,-52.760,-179.319,6.448,148.975
C01532=1153.385,86.339,-52.742,-179.321,6.447,148.975
C01533=1153.390,86.089,-52.725,-179.324,6.445,148.976
C01534=1153.395,85.840,-52.707,-179.327,6.444,148.976
C01535=1153.400,85.591,-52.690,-179.329,6.443,148.976
C01536=1153.405,85.341,-52.672,-179.332,6.442,148.977
C01537=1153.410,85.092,-52.655,-179.335,6.440,148.978
C01538=1153.415,84.842,-52.637,-179.337,6.439,148.978
C01539=1153.420,84.594,-52.620,-179.340,6.438,148.979
C01540=1153.425,84.344,-52.603,-179.343,6.436,148.979
C01541=1153.430,84.095,-52.585,-179.345,6.435,148.979
C01542=1153.434,83.846,-52.568,-179.348,6.433,148.980
C01543=1153.440,83.596,-52.551,-179.351,6.432,148.981
C01544=1153.444,83.347,-52.533,-179.353,6.431,148.981
C01545=1153.449,83.097,-52.516,-179.356,6.430,148.981
C01546=1153.454,82.848,-52.498,-179.359,6.428,148.982
C01547=1153.459,82.598,-52.481,-179.361,6.427,148.982
C01548=1153.464,82.349,-52.463,-179.364,6.426,148.983
C01549=1153.469,82.100,-52.446,-179.367,6.424,148.984
C01550=1153.474,81.851,-52.429,-179.369,6.424,148.984
C01551=1153.478,81.602,-52.412,-179.372,6.422,148.984
C01552=1153.484,81.352,-52.395,-179.375,6.421,148.985
C01553=1153.489,81.102,-52.377,-179.378,6.420,148.985
C01554=1153.493,80.853,-52.360,-179.380,6.418,148.986
C01555=1153.498,80.604,-52.343,-179.383,6.416,148.986
C01556=1153.504,80.354,-52.326,-179.386,6.416,148.987
C01557=1153.509,80.086,-52.308,-179.388,6.414,148.987
C01558=1153.514,79.818,-52.288,-179.392,6.413,148.988
C01559=1153.520,79.549,-52.270,-179.394,6.411,148.988
C01560=1153.524,79.281,-52.252,-179.398,6.410,148.989
C01561=1153.530,79.031,-52.235,-179.400,6.409,148.990
C01562=1153.534,78.782,-52.218,-179.402,6.407,148.990
C01563=1153.540,78.533,-52.200,-179.406,6.406,148.991
C01564=1153.544,78.284,-52.184,-179.408,6.405,148.991
C01565=1153.549,78.034,-52.166,-179.411,6.403,148.992
C01566=1153.555,77.784,-52.149,-179.414,6.402,148.992
C01567=1153.559,77.535,-52.132,-179.416,6.401,148.993
C01568=1153.565,77.286,-52.115,-179.419,6.400,148.993
C01569=1153.569,77.037,-52.098,-179.422,6.398,148.994
C01570=1153.574,76.787,-52.081,-179.424,6.397,148.994
C01571=1153.579,76.537,-52.064,-179.427,6.396,148.995
C01572=1153.584,76.289,-52.047,-179.429,6.395,148.995
C01573=1153.589,76.039,-52.030,-179.432,6.394,148.996
C01574=1153.594,75.790,-52.013,-179.435,6.392,148.996
C01575=1153.598,75.540,-51.996,-179.438,6.391,148.997
C01576=1153.604,75.291,-51.980,-179.440,6.390,148.997
C01577=1153.609,75.042,-51.962,-179.442,6.389,148.998
C01578=1153.613,74.792,-51.946,-179.446,6.388,148.998
C01579=1153.618,74.542,-51.928,-179.448,6.386,148.999
C01580=1153.624,74.293,-51.912,-179.451,6.385,148.999
C01581=1153.628,74.044,-51.894,-179.454,6.384,149.000
C01582=1153.633,73.795,-51.877,-179.456,6.382,149.000
C01583=1153.638,73.545,-51.860,-179.459,6.381,149.001
C01584=1153.643,73.296,-51.844,-179.462,6.380,149.001
C01585=1153.648,73.047,-51.827,-179.464,6.379,149.002
C01586=1153.653,72.797,-51.810,-179.467,6.378,149.002
C01587=1153.658,72.548,-51.794,-179.470,6.376,149.003
C01588=1153.662,72.299,-51.777,-179.472,6.375,149.003
C01589=1153.668,72.049,-51.760,-179.475,6.374,149.004
C01590=1153.673,71.800,-51.743,-179.477,6.373,149.004
C01591=1153.678,71.550,-51.726,-179.480,6.371,149.005
C01592=1153.682,71.301,-51.709,-179.483,6.371,149.005
C01593=1153.687,71.051,-51.693,-179.486,6.369,149.006
C01594=1153.693,70.802,-51.676,-179.488,6.367,149.006
C01595=1153.697,70.553,-51.659,-179.491,6.367,149.007
C01596=1153.703,70.303,-51.644,-179.494,6.365,149.007
C01597=1153.708,70.054,-51.626,-179.496,6.364,149.008
C01598=1153.712,69.804,-51.610,-179.499,6.363,149.008
C01599=1153.717,69.555,-51.593,-179.502,6.361,149.009
C01600=1153.723,69.305,-51.576,-179.504,6.361,149.009
C01601=1153.727,69.056,-51.559,-179.507,6.359,149.010
C01602=1153.732,68.807,-51.543,-179.509,6.358,149.010
C01603=1153.737,68.558,-51.527,-179.513,6.357,149.011
C01604=1153.742,68.307,-51.510,-179.515,6.356,149.011
C01605=1153.747,68.059,-51.494,-179.517,6.355,149.012
C01606=1153.752,67.809,-51.477,-179.520,6.354,149.013
C01607=1153.757,67.560,-51.461,-179.523,6.352,149.013
C01608=1153.762,67.310,-51.443,-179.526,6.351,149.013
C01609=1153.767,67.061,-51.427,-179.528,6.350,149.014
C01610=1153.772,66.812,-51.411,-179.531,6.349,149.015
C01611=1153.776,66.562,-51.395,-179.534,6.348,149.015
C01612=1153.782,66.313,-51.378,-179.536,6.346,149.016
C01613=1153.787,66.064,-51.361,-179.538,6.346,149.016
C01614=1153.791,65.813,-51.345,-179.542,6.344,149.017
C01615=1153.797,65.565,-51.329,-179.544,6.343,149.017
C01616=1153.801,65.315,-51.312,-179.547,6.342,149.018
C01617=1153.807,65.066,-51.295,-179.550,6.340,149.018
C01618=1153.812,64.816,-51.279,-179.552,6.340,149.019
C01619=1153.817,64.567,-51.263,-179.555,6.338,149.019
C01620=1153.821,64.318,-51.246,-179.557,6.337,149.020
C01621=1153.826,64.068,-51.230,-179.560,6.336,149.020
C01622=1153.831,63.819,-51.214,-179.563,6.335,149.021
C01623=1153.836,63.569,-51.197,-179.565,6.334,149.021
C01624=1153.842,63.320,-51.181,-179.568,6.333,149.022
C01625=1153.846,63.070,-51.164,-179.571,6.331,149.022
C01626=1153.851,62.821,-51.148,-179.573,6.331,149.023
C01627=1153.856,62.571,-51.132,-179.576,6.329,149.023
C01628=1153.861,62.322,-51.116,-179.578,6.328,149.024
C01629=1153.866,62.072,-51.100,-179.581,6.327,149.024
C01630=1153.871,61.824,-51.084,-179.584,6.326,149.025
C01631=1153.875,61.574,-51.067,-179.587,6.325,149.025
C01632=1153.881,61.325,-51.051,-179.590,6.323,149.026
C01633=1153.886,61.075,-51.034,-179.592,6.322,149.027
C01634=1153.891,60.825,-51.018,-179.595,6.321,149.027
C01635=1153.896,60.576,-51.002,-179.597,6.320,149.028
C01636=1153.901,60.327,-50.986,-179.600,6.319,149.028
C01637=1153.906,60.077,-50.970,-179.603,6.318,149.029
C01638=1153.911,59.828,-50.954,-179.605,6.317,149.029
C01639=1153.916,59.578,-50.937,-179.608,6.316,149.030
C01640=1153.921,59.329,-50.922,-179.611,6.314,149.030
C01641=1153.926,59.079,-50.905,-179.613,6.314,149.031
C01642=1153.931,58.830,-50.889,-179.616,6.312,149.031
C01643=1153.936,58.581,-50.873,-179.618,6.311,149.032
C01644=1153.941,58.331,-50.857,-179.621,6.310,149.032
C01645=1153.946,58.082,-50.841,-179.624,6.309,149.033
C01646=1153.951,57.832,-50.825,-179.626,6.308,149.033
C01647=1153.956,57.583,-50.809,-179.629,6.307,149.034
C01648=1153.960,57.333,-50.793,-179.632,6.305,149.034
C01649=1153.966,57.084,-50.777,-179.634,6.305,149.035
C01650=1153.970,56.834,-50.760,-179.637,6.303,149.036
C01651=1153.976,56.585,-50.745,-179.639,6.302,149.036
C01652=1153.981,56.336,-50.729,-179.643,6.301,149.037
C01653=1153.986,56.086,-50.713,-179.645,6.300,149.037
C01654=1153.991,55.837,-50.697,-179.647,6.299,149.038
C01655=1153.995,55.587,-50.680,-179.650,6.298,149.038
C01656=1154.000,55.338,-50.665,-179.652,6.297,149.039
C01657=1154.006,55.089,-50.650,-179.656,6.296,149.039
C01658=1154.010,54.839,-50.633,-179.658,6.295,149.040
C01659=1154.015,54.590,-50.617,-179.660,6.293,149.040
C01660=1154.021,54.340,-50.602,-179.663,6.293,149.041
C01661=1154.026,54.071,-50.585,-179.666,6.291,149.041
C01662=1154.031,53.803,-50.567,-179.669,6.290,149.042
C01663=1154.037,53.534,-50.550,-179.672,6.290,149.043
C01664=1154.042,53.266,-50.533,-179.674,6.288,149.043
C01665=1154.047,53.016,-50.517,-179.677,6.287,149.044
C01666=1154.052,52.767,-50.501,-179.680,6.286,149.044
C01667=1154.057,52.518,-50.486,-179.682,6.285,149.045
C01668=1154.062,52.268,-50.470,-179.685,6.284,149.045
C01669=1154.067,52.018,-50.455,-179.687,6.283,149.046
C01670=1154.072,51.770,-50.438,-179.691,6.281,149.046
C01671=1154.077,51.519,-50.422,-179.693,6.281,149.047
C01672=1154.082,51.270,-50.407,-179.696,6.279,149.048
C01673=1154.087,51.021,-50.392,-179.698,6.278,149.048
C01674=1154.092,50.771,-50.376,-179.700,6.278,149.048
C01675=1154.097,50.522,-50.360,-179.704,6.276,149.049
C01676=1154.102,50.273,-50.344,-179.706,6.275,149.050
C01677=1154.107,50.024,-50.329,-179.709,6.274,149.050
C01678=1154.112,49.773,-50.313,-179.711,6.273,149.051
C01679=1154.117,49.524,-50.297,-179.714,6.272,149.051
C01680=1154.122,49.275,-50.282,-179.716,6.271,149.052
C01681=1154.127,49.025,-50.266,-179.719,6.270,149.052
C01682=1154.132,48.775,-50.251,-179.722,6.269,149.053
C01683=1154.137,48.526,-50.235,-179.724,6.268,149.053
C01684=1154.142,48.277,-50.219,-179.727,6.267,149.054
C01685=1154.146,48.028,-50.204,-179.729,6.266,149.054
C01686=1154.152,47.778,-50.188,-179.732,6.264,149.055
C01687=1154.157,47.529,-50.172,-179.735,6.264,149.056
C01688=1154.163,47.279,-50.157,-179.738,6.262,149.056
C01689=1154.167,47.030,-50.142,-179.740,6.262,149.057
C01690=1154.172,46.780,-50.126,-179.742,6.261,149.057
C01691=1154.177,46.531,-50.110,-179.746,6.260,149.058
C01692=1154.182,46.282,-50.095,-179.748,6.259,149.058
C01693=1154.187,46.032,-50.079,-179.751,6.258,149.059
C01694=1154.192,45.782,-50.064,-179.753,6.257,149.059
C01695=1154.197,45.533,-50.049,-179.755,6.256,149.060
C01696=1154.202,45.284,-50.033,-179.759,6.255,149.060
C01697=1154.207,45.033,-50.017,-179.761,6.254,149.061
C01698=1154.212,44.784,-50.002,-179.764,6.252,149.062
C01699=1154.217,44.535,-49.987,-179.766,6.252,149.062
C01700=1154.223,44.285,-49.972,-179.769,6.250,149.063
C01701=1154.227,44.036,-49.957,-179.771,6.249,149.063
C01702=1154.232,43.786,-49.941,-179.774,6.249,149.064
C01703=1154.237,43.537,-49.926,-179.777,6.247,149.064
C01704=1154.242,43.287,-49.910,-179.779,6.246,149.065
C01705=1154.248,43.038,-49.895,-179.782,6.245,149.065
C01706=1154.252,42.789,-49.880,-179.784,6.244,149.066
C01707=1154.258,42.539,-49.864,-179.787,6.244,149.066
C01708=1154.262,42.289,-49.850,-179.790,6.242,149.067
C01709=1154.267,42.040,-49.834,-179.792,6.242,149.068
C01710=1154.273,41.790,-49.818,-179.795,6.241,149.068
C01711=1154.277,41.541,-49.803,-179.797,6.239,149.068
C01712=1154.283,41.292,-49.788,-179.800,6.239,149.069
C01713=1154.287,41.043,-49.773,-179.803,6.237,149.070
C01714=1154.293,40.793,-49.758,-179.805,6.237,149.070
C01715=1154.297,40.543,-49.743,-179.808,6.236,149.071
C01716=1154.303,40.293,-49.727,-179.811,6.235,149.071
C01717=1154.307,40.044,-49.712,-179.813,6.234,149.072
C01718=1154.313,39.794,-49.697,-179.816,6.233,149.073
C01719=1154.318,39.545,-49.682,-179.818,6.232,149.073
C01720=1154.323,39.296,-49.667,-179.821,6.231,149.074
C01721=1154.328,39.047,-49.652,-179.824,6.229,149.074
C01722=1154.333,38.797,-49.637,-179.826,6.229,149.075
C01723=1154.337,38.547,-49.621,-179.829,6.228,149.075
C01724=1154.343,38.297,-49.606,-179.831,6.226,149.076
C01725=1154.348,38.048,-49.591,-179.834,6.226,149.076
C01726=1154.353,37.798,-49.576,-179.836,6.225,149.077
C01727=1154.358,37.549,-49.561,-179.839,6.224,149.077
C01728=1154.363,37.299,-49.546,-179.841,6.223,149.078
C01729=1154.368,37.050,-49.531,-179.844,6.223,149.079
C01730=1154.373,36.801,-49.515,-179.847,6.221,149.079
C01731=1154.378,36.551,-49.501,-179.850,6.220,149.080
C01732=1154.383,36.302,-49.486,-179.852,6.219,149.080
C01733=1154.388,36.053,-49.471,-179.854,6.218,149.081
C01734=1154.393,35.803,-49.456,-179.857,6.218,149.081
C01735=1154.399,35.553,-49.441,-179.860,6.216,149.082
C01736=1154.404,35.304,-49.426,-179.863,6.215,149.082
C01737=1154.408,35.055,-49.411,-179.865,6.215,149.083
C01738=1154.414,34.805,-49.397,-179.868,6.213,149.084
C01739=1154.419,34.556,-49.382,-179.870,6.212,149.084
C01740=1154.424,34.306,-49.366,-179.873,6.212,149.085
C01741=1154.428,34.056,-49.351,-179.875,6.210,149.085
C01742=1154.433,33.807,-49.336,-179.878,6.210,149.086
C01743=1154.439,33.557,-49.321,-179.880,6.209,149.086
C01744=1154.443,33.308,-49.306,-179.884,6.208,149.087
C01745=1154.448,33.058,-49.292,-179.886,6.207,149.087
C01746=1154.454,32.808,-49.277,-179.888,6.206,149.088
C01747=1154.459,32.559,-49.262,-179.891,6.205,149.088
C01748=1154.463,32.310,-49.247,-179.893,6.204,149.089
C01749=1154.469,32.060,-49.232,-179.896,6.203,149.090
C01750=1154.474,31.810,-49.217,-179.899,6.202,149.090
C01751=1154.479,31.561,-49.203,-179.901,6.201,149.091
C01752=1154.485,31.311,-49.189,-179.903,6.201,149.091
C01753=1154.490,31.062,-49.174,-179.907,6.199,149.092
C01754=1154.495,30.813,-49.159,-179.909,6.198,149.092
C01755=1154.499,30.564,-49.144,-179.911,6.198,149.093
C01756=1154.505,30.314,-49.130,-179.914,6.197,149.093
C01757=1154.510,30.064,-49.115,-179.917,6.196,149.094
C01758=1154.515,29.815,-49.100,-179.919,6.195,149.095
C01759=1154.520,29.565,-49.086,-179.922,6.195,149.095
C01760=1154.525,29.316,-49.070,-179.924,6.193,149.096
C01761=1154.530,29.066,-49.056,-179.927,6.192,149.096
C01762=1154.535,28.816,-49.042,-179.929,6.192,149.097
C01763=1154.539,28.567,-49.027,-179.932,6.190,149.097
C01764=1154.545,28.317,-49.012,-179.935,6.190,149.098
C01765=1154.550,28.048,-48.996,-179.937,6.189,149.099
C01766=1154.555,27.779,-48.981,-179.940,6.187,149.099
C01767=1154.561,27.511,-48.965,-179.943,6.187,149.100
C01768=1154.567,27.241,-48.949,-179.946,6.186,149.100
C01769=1154.572,26.993,-48.935,-179.948,6.185,149.101
C01770=1154.577,26.743,-48.920,-179.951,6.184,149.102
C01771=1154.582,26.493,-48.906,-179.954,6.183,149.102
C01772=1154.587,26.243,-48.892,-179.956,6.182,149.102
C01773=1154.592,25.994,-48.876,-179.958,6.181,149.103
C01774=1154.597,25.744,-48.862,-179.961,6.181,149.104
C01775=1154.602,25.495,-48.848,-179.964,6.179,149.104
C01776=1154.607,25.245,-48.833,-179.966,6.179,149.105
C01777=1154.612,24.997,-48.819,-179.969,6.178,149.105
C01778=1154.617,24.747,-48.804,-179.971,6.176,149.106
C01779=1154.622,24.497,-48.790,-179.974,6.176,149.107
C01780=1154.628,24.247,-48.775,-179.976,6.175,149.107
C01781=1154.633,23.997,-48.761,-179.979,6.175,149.108
C01782=1154.638,23.748,-48.747,-179.982,6.173,149.108
C01783=1154.642,23.499,-48.732,-179.984,6.173,149.109
C01784=1154.648,23.250,-48.718,-179.986,6.172,149.109
C01785=1154.653,23.000,-48.704,-179.989,6.171,149.110
C01786=1154.658,22.750,-48.689,-179.992,6.170,149.110
C01787=1154.663,22.500,-48.675,-179.994,6.169,149.111
C01788=1154.668,22.251,-48.661,-179.997,6.168,149.112
C01789=1154.673,22.001,-48.646,-180.000,6.167,149.112
C01790=1154.678,21.753,-48.632,179.998,6.166,149.113
C01791=1154.683,21.503,-48.618,179.995,6.166,149.113
C01792=1154.688,21.253,-48.603,179.993,6.165,149.114
C01793=1154.693,21.004,-48.589,179.990,6.164,149.115
C01794=1154.698,20.754,-48.575,179.988,6.163,149.115
C01795=1154.704,20.504,-48.560,179.985,6.162,149.116
C01796=1154.709,20.255,-48.546,179.983,6.162,149.116
C01797=1154.714,20.005,-48.532,179.980,6.160,149.117
C01798=1154.719,19.755,-48.517,179.978,6.159,149.117
C01799=1154.724,19.506,-48.503,179.975,6.159,149.118
C01800=1154.730,19.257,-48.489,179.973,6.158,149.118
C01801=1154.735,19.007,-48.475,179.971,6.157,149.119
C01802=1154.739,18.757,-48.461,179.967,6.156,149.120
C01803=1154.744,18.508,-48.447,179.965,6.155,149.120
C01804=1154.749,18.259,-48.433,179.962,6.155,149.121
C01805=1154.754,18.009,-48.419,179.960,6.154,149.121
C01806=1154.759,17.759,-48.405,179.957,6.153,149.122
C01807=1154.764,17.510,-48.390,179.955,6.152,149.122
C01808=1154.770,17.261,-48.376,179.952,6.151,149.123
C01809=1154.775,17.011,-48.362,179.950,6.151,149.123
C01810=1154.780,16.761,-48.348,179.947,6.149,149.124
C01811=1154.785,16.511,-48.334,179.945,6.149,149.125
C01812=1154.790,16.262,-48.320,179.942,6.148,149.125
C01813=1154.795,16.012,-48.306,179.940,6.147,149.126
C01814=1154.800,15.762,-48.292,179.937,6.147,149.126
C01815=1154.806,15.513,-48.278,179.934,6.145,149.127
C01816=1154.811,15.264,-48.264,179.932,6.145,149.128
